METHOD PublishReceived : BOOL
  VAR_INPUT
    Data : MQTT.CALLBACK_DATA;  (* Collection of recived Data *)
  END_VAR
  VAR
    sSubTopic : STRING;
    NodeNumber : STRING;
    sNodeRegister : STRING;
    iWritePos : INT;  (* 1-based position of '/write/' within sSubTopic; 0 when it is absent. *)
  END_VAR
                  //first check if Mqtt is initialized, otherwise do nothing
IF NOT(bInitMqttDone) THEN
	//mark the interface call from the collector as done
	PublishReceived := TRUE;
//check if the packet is for this FB
ELSIF sMQTTSubscribeTopic = LEFT(Data.TopicOut^, LEN(sMQTTSubscribeTopic)) THEN
	//mark the interface call from the collector as done
	PublishReceived := TRUE;
	// process the data
	(* Parse by delimiter rather than by fixed width. The old code took the last
	   nine characters and then one character each for the node and the register,
	   so a command on '.../12/write/3' parsed as node 2 - a write silently aimed
	   at a different physical device. This block supports afbNodes 2..30. *)
	sSubTopic := RIGHT(Data.TopicOut^, LEN(Data.TopicOut^) - LEN(sMQTTSubscribeTopic));
	iWritePos := FIND(sSubTopic, '/write/');

	IF iWritePos >= 3 THEN
		// sSubTopic is '/<node>/write/<register>', so the node digits occupy
		// positions 2..iWritePos-1 and the register is everything past '/write/'.
		NodeNumber := MID(sSubTopic, iWritePos - 2, 2);
		sNodeRegister := RIGHT(sSubTopic, LEN(sSubTopic) - (iWritePos + 6));
	ELSE
		NodeNumber := '';
		sNodeRegister := '';
	END_IF

	(* A payload may be negative: -1 on a target register is how a Ducobox is told
	   to stop overriding and return to automatic, and the box's own target entity
	   is announced with a minimum of -1 for exactly that. The sign is taken off
	   before the digits are checked - so whether IS_NUM accepts a leading minus
	   does not matter - and put back through INT_TO_WORD, whose two's complement
	   is what the device reads back as -1. STRING_TO_WORD on '-1' does not. *)
	sPayload := Data.PayloadString^;
	bNegative := LEFT(sPayload, 1) = '-';
	IF bNegative THEN
		sDigits := RIGHT(sPayload, LEN(sPayload) - 1);
	ELSE
		sDigits := sPayload;
	END_IF

	IF iWritePos >= 3 AND
		OSCAT_BASIC.IS_NUM(NodeNumber) AND
		OSCAT_BASIC.IS_NUM(sNodeRegister) AND
		OSCAT_BASIC.IS_NUM(sDigits) AND
		(* 1 is the box itself, 2 and up are its components. The box is written
		   exactly like a component - its registers start at 10, which is what
		   index 1 gives - and InitMqttDiscovery announces three numbers and five
		   buttons for it. Requiring 2 here left every one of those controls inert,
		   and silently: falling through this guard looks identical to a topic
		   meant for some other device. *)
		STRING_TO_UINT(NodeNumber) >= 1 AND
		STRING_TO_UINT(NodeNumber) < THIS^.uiNodePointer THEN
			stWriteStep.Address := (STRING_TO_UINT(NodeNumber) * 10) + STRING_TO_UINT(sNodeRegister);
			IF bNegative THEN
				stWriteStep.Data[0] := INT_TO_WORD(-1 * STRING_TO_INT(sDigits));
			ELSE
				stWriteStep.Data[0] := STRING_TO_WORD(sDigits);
			END_IF
			sWriteQuerySuffix := sSubTopic;
			sWriteQueryPayload := Data.PayloadString^;
			bWriteQueryReady := TRUE;
	END_IF
END_IF
                
END_METHOD

METHOD AddNode : BOOL
  VAR_INPUT
    FriendlyName : STRING(GVL_MQTT.MQTT_SUFFIX_LEN);  (* Name of the room this component serves. *)
    DataPollingInterval : TIME;
  END_VAR
                  (* afbNodes is ARRAY[2..30]. Without this bound the 30th call wrote past the end of
   it, and the unassigned return value left the caller unable to notice. *)
IF uiNodePointer <= 30 THEN
	THIS^.afbNodes[uiNodePointer].InitNode(
		DeviceAddress := THIS^.stMasterStep.DeviceId,
		NodeNumber := uiNodePointer - 1,
		FriendlyName := FriendlyName,
		DataPollingInterval := DataPollingInterval
	);

	uiNodePointer := uiNodePointer + 1;
	AddNode := TRUE;
ELSE
	AddNode := FALSE;
END_IF

                
END_METHOD

METHOD BuildTransaction : INT
  VAR_INPUT
    pSteps : POINTER TO A_RS485_STEP_LIST;
  END_VAR
  VAR
    iN : INT;
    iK : INT;
    iI : INT;
  END_VAR
                  iN := 0;

IF bWriteQueryReady THEN
	bWriteQueryReady := FALSE;

	(* Write, then read the same register straight back, with the bus held
	   across both. What this block used to do was publish the payload it had
	   just sent, as though sending it were proof - so Home Assistant showed a
	   value the Ducobox might never have taken. AbortOnError on the write is
	   what stops the read-back running, and therefore stops anything being
	   published, when the write itself fails. *)
	pSteps^[iN]				:= stWriteStep;
	pSteps^[iN].AbortOnError	:= TRUE;
	aiStepMap[iN]				:= 2;
	iN						:= iN + 1;

	stReadBackStep.DeviceId		:= stWriteStep.DeviceId;
	(* Function 3: the register was written as a holding register, so that is
	   where it reads back from. If a Ducobox turns out to mirror these into the
	   input register space instead, this is the one line that changes. *)
	stReadBackStep.FunctionCode	:= 3;
	stReadBackStep.Address		:= stWriteStep.Address;
	stReadBackStep.Quantity		:= 1;

	pSteps^[iN]	:= stReadBackStep;
	aiStepMap[iN]	:= 3;
	iN			:= iN + 1;
END_IF

IF fbTimerData.Q THEN
	fbTimerData.IN	:= FALSE;
	pSteps^[iN]		:= stMasterStep;
	aiStepMap[iN]		:= 1;
	iN				:= iN + 1;
END_IF

(* One node per transaction, taken in turn from iNodeCursor. *)
FOR iK := 0 TO 28 DO
	iI := 2 + ((iNodeCursor - 2 + iK) MOD 29);
	IF iI < UINT_TO_INT(uiNodePointer) THEN
		IF afbNodes[iI].RequestBusTime() THEN
			pSteps^[iN]	:= afbNodes[iI].GetStep();
			aiStepMap[iN]	:= 10 + iI;
			iN			:= iN + 1;
			iNodeCursor	:= 2 + ((iI - 1) MOD 29);
			EXIT;
		END_IF
	END_IF
END_FOR

(* The zone read, at most one per transaction and only until each node has
   answered once. It rides behind the value read rather than competing with it,
   and it is a step of its own because read parameters 6..8 are undefined and the
   box rejects a span that crosses them. *)
FOR iK := 2 TO 30 DO
	IF iK < UINT_TO_INT(uiNodePointer) THEN
		IF afbNodes[iK].RequestLocation() THEN
			(* GetLocationStep answers with a zero-filled step if its retry clock
			   lapsed since RequestLocation was asked. Quantity 0 is not a Modbus
			   request: it fails locally, never reaches the bus, and so never shows
			   in the counters - while still counting as a failed step here. *)
			stLocStep := afbNodes[iK].GetLocationStep();
			IF stLocStep.Quantity > 0 THEN
				pSteps^[iN]	:= stLocStep;
				aiStepMap[iN]	:= 50 + iK;
				iN			:= iN + 1;
			END_IF
			EXIT;
		END_IF
	END_IF
END_FOR

(* One setting register per transaction, the box's own first. Deliberately
   last and one at a time: this is refresh traffic, it must never crowd out a
   command or a measurement, and reading a span would cross registers that are
   undefined on some component types. *)
IF bBoxSettingsDue THEN
	iBoxSettingsPending := -1;
	FOR iB := iBoxSettingsCursor TO 9 DO
		IF (wBoxSettingsMask AND SHL(WORD#1, INT_TO_BYTE(iB))) <> 0 THEN
			iBoxSettingsPending := iB;
			iBoxSettingsCursor := iB + 1;
			EXIT;
		END_IF
	END_FOR

	IF iBoxSettingsPending >= 0 THEN
		stBoxSettingsStep.Address := 10 + INT_TO_UINT(iBoxSettingsPending);
		pSteps^[iN]	:= stBoxSettingsStep;
		aiStepMap[iN]	:= 4;
		iN			:= iN + 1;
	ELSE
		bBoxSettingsDue := FALSE;
	END_IF
ELSE
	FOR iK := 2 TO 30 DO
		IF iK < UINT_TO_INT(uiNodePointer) THEN
			IF afbNodes[iK].RequestSettings() THEN
				stLocStep := afbNodes[iK].GetSettingsStep();
				IF stLocStep.Quantity > 0 THEN
					pSteps^[iN]	:= stLocStep;
					aiStepMap[iN]	:= 100 + iK;
					iN			:= iN + 1;
				END_IF
				EXIT;
			END_IF
		END_IF
	END_FOR
END_IF

(* Whether this transaction carried anything whose failure would really mean
   the box is unreachable: the master read, or a node's measurements. A lone
   zone read does not qualify. *)
bTxHadRequiredStep := FALSE;
FOR iK := 0 TO iN - 1 DO
	IF (aiStepMap[iK] = 1) OR ((aiStepMap[iK] >= 12) AND (aiStepMap[iK] <= 40)) THEN
		bTxHadRequiredStep := TRUE;
	END_IF
END_FOR

BuildTransaction := iN;

                
END_METHOD

METHOD HasWork : E_RS485_WORK_LEVEL
  VAR
    iK : INT;
  END_VAR
                  (* Pure predicate. afbNodes[].RequestBusTime is one too, so asking them here costs
   nothing and cannot disturb anything - which is the reason the node kept that
   method while the parent's own version was replaced. *)
IF NOT bInitRS485Done THEN
	HasWork := E_RS485_WORK_LEVEL.NONE;
	RETURN;
END_IF

IF bWriteQueryReady THEN
	(* Somebody is waiting on this: it arrived over MQTT, from Home Assistant or
	   a person. Ahead of routine polling, but still round-robin against other
	   devices' commands. *)
	HasWork := E_RS485_WORK_LEVEL.COMMAND;
	RETURN;
END_IF

IF fbTimerData.Q THEN
	HasWork := E_RS485_WORK_LEVEL.POLL;
	RETURN;
END_IF

IF bBoxSettingsDue THEN
	(* Refresh traffic, so it ranks with polling rather than with a command. *)
	HasWork := E_RS485_WORK_LEVEL.POLL;
	RETURN;
END_IF

HasWork := E_RS485_WORK_LEVEL.NONE;
FOR iK := 2 TO 30 DO
	IF iK < UINT_TO_INT(uiNodePointer) THEN
		(* RequestLocation counts as work: without it a node that has answered its
		   values but not its zone would never get another transaction built. *)
		IF afbNodes[iK].RequestBusTime() OR afbNodes[iK].RequestLocation()
			OR afbNodes[iK].RequestSettings() THEN
			HasWork := E_RS485_WORK_LEVEL.POLL;
			RETURN;
		END_IF
	END_IF
END_FOR

                
END_METHOD

METHOD OnStepResult
  VAR_INPUT
    StepIndex : INT;
    Failed : BOOL;
    pData : POINTER TO A_RS485_READ_BUFFER;
    Count : INT;
  END_VAR
  VAR
    iStepKind : INT;
  END_VAR
                  IF StepIndex < 0 OR StepIndex > DINT_TO_INT(UPPER_BOUND(aiStepMap, 1)) THEN
	RETURN;
END_IF

iStepKind := aiStepMap[StepIndex];

IF iStepKind = 1 THEN
	(* Master unit *)
	THIS^.Error := Failed;
	THIS^.fbTimerData.IN := TRUE;
	IF NOT Failed AND Count >= 6 THEN
		(* Publish only what moved. The box answers with the same six values poll
		   after poll - on the bench that was 126 identical messages in 100 seconds
		   against one or two from each node - and volume on this task is what made
		   the publish-queue race fire constantly before the queue got lanes.

		   Topics are not retained, so a value that never moves would never reach a
		   reconnecting Home Assistant; the refresh in the body forces a full
		   publish periodically regardless. *)
		bMasterChanged := NOT bMasterPublished OR bRefreshDue;
		FOR iMasterChk := 0 TO 5 DO
			IF pData^[iMasterChk] <> awLastMaster[iMasterChk] THEN
				bMasterChanged := TRUE;
			END_IF
			awLastMaster[iMasterChk] := pData^[iMasterChk];
		END_FOR

		IF bMasterChanged THEN
			bMasterPublished := TRUE;
			bRefreshDue := FALSE;
			PubMqttMessage(Suffix := '/1/TYPE', Data := F_DUCO_TYPE_TEXT(F_DUCO_NODE_TYPE(pData^[0])));
			PubMqttMessage(Suffix := '/1/STATUS', Data := F_DUCO_STATUS_TEXT(pData^[1]));
			PubMqttMessage(Suffix := '/1/POS', Data := WORD_TO_STRING(pData^[2]));
			(* Focus-specific: on this box read parameters 3, 4 and 5 are the current,
			   average and maximum power in watts. Another DucoBox answers the same
			   addresses with a different set, which is why this block is named. *)
			PubMqttMessage(Suffix := '/1/PWR', Data := WORD_TO_STRING(pData^[3]));
			PubMqttMessage(Suffix := '/1/PWR_AVG', Data := WORD_TO_STRING(pData^[4]));
			PubMqttMessage(Suffix := '/1/PWR_MAX', Data := WORD_TO_STRING(pData^[5]));
		END_IF
	END_IF

ELSIF iStepKind = 2 THEN
	(* The write. Deliberately publishes nothing: the value is only news once
	   the device has been read back and agrees. *)
	THIS^.Error := Failed;

ELSIF iStepKind = 3 THEN
	(* The read-back. This is the value the device actually holds, which is the
	   whole point of pairing the two. *)
	IF NOT Failed AND Count >= 1 THEN
		(* Suffix already begins with '/', so this leading one doubles it. Kept
		   as it was: the topic is what Home Assistant is already subscribed to,
		   and it cannot be re-checked without a Ducobox on the bench. *)
		(* One slash, not two. The suffix already begins with one, and the doubled
   topic was only harmless while nothing subscribed to it. The number and
   switch entities now take their state from here, so it has to be the topic
   their discovery config names. *)
PubMqttMessage(Suffix := sWriteQuerySuffix, Data := INT_TO_STRING(WORD_TO_INT(pData^[0])));
	END_IF

ELSIF iStepKind = 4 THEN
	(* The box's own setting, read back so its entity has a value before anybody
	   sets one. Signed for the same reason the write path is: -1 is a real
	   value here, meaning the box is not overriding. *)
	IF NOT Failed AND Count >= 1 AND iBoxSettingsPending >= 0 THEN
		PubMqttMessage(
			Suffix := CONCAT('/1/write/', INT_TO_STRING(iBoxSettingsPending)),
			Data := INT_TO_STRING(WORD_TO_INT(pData^[0])));
	END_IF
	iBoxSettingsPending := -1;

ELSIF iStepKind >= 12 AND iStepKind <= 40 THEN
	afbNodes[iStepKind - 10].OnStepResult(Failed := Failed, pData := pData, Count := Count);

ELSIF iStepKind >= 102 AND iStepKind <= 130 THEN
	(* 100 + node index: a setting register read back. A separate kind again,
	   because it lands in its own method and carries one register. *)
	afbNodes[iStepKind - 100].OnSettingsResult(Failed := Failed, pData := pData, Count := Count);

ELSIF iStepKind >= 52 AND iStepKind <= 80 THEN
	(* 50 + node index: the zone read. A separate kind from 10 + index because the
	   two steps carry different registers and land in different methods. *)
	afbNodes[iStepKind - 50].OnLocationResult(Failed := Failed, pData := pData, Count := Count);
END_IF

                
END_METHOD

METHOD OnTransactionDone
  VAR_INPUT
    StepsRun : INT;
    Failures : INT;
  END_VAR
                  (* Count, do not decide - and record what was actually seen.

   A single transaction is far too small a sample to condemn a device on: this
   bus interleaves the master read, one node's measurements, an optional zone
   read and any write that has arrived, and the mix differs every time. The
   verdict is taken on a heartbeat in the body instead. *)
uiTxCalls := uiTxCalls + 1;
iLastStepsRun := StepsRun;
iLastFailures := Failures;

IF StepsRun > 0 AND bTxHadRequiredStep THEN
	uiTxSeen := uiTxSeen + 1;
	IF Failures < StepsRun THEN
		uiTxOk := uiTxOk + 1;
	END_IF
END_IF

                
END_METHOD

(* Nothing to commission on this device. See I_RS485_DEVICE.GetCommissioning. *)
METHOD GetCommissioning : BOOL
  VAR_INPUT
    BusBaudrate : UDINT;
    pRequest : POINTER TO ST_RS485_COMMISSION_REQUEST;
  END_VAR
                  (* Nothing to commission. This device is configured on the device itself - switches,
   a display, or a factory setting that already matches this bus - so it answers at
   whatever the bus runs at and there is nothing for the commissioner to write.

   Which is the ordinary case: the cost of the whole mechanism, for a device like
   this one, is this method call once at bStartup. *)
GetCommissioning := FALSE;

                
END_METHOD

(* Announce the box and, as the bus reports what they are, every component on it. Call once at startup, after InitMqtt. *)
METHOD InitMqttDiscovery
  VAR_INPUT
    DeviceName : STRING(50);
    overruleId : STRING(255);
  END_VAR
  VAR
    sLabel : STRING(GVL_MQTT.MQTT_SUFFIX_LEN);
    sOut : STRING(GVL_MQTT.MQTT_TOPIC_LEN);
    sCmd : STRING(GVL_MQTT.MQTT_TOPIC_LEN);
  END_VAR
                  (* The box itself is node 1. Its own device; each component announces its own
   as the bus reports what it is, from the sweep in the body. *)
IF bInitMqttDone AND NOT bInitMqttDiscoveryDone THEN
	bInitMqttDiscoveryDone := TRUE;
	sDeviceId := SUPER^.ResolveEntityId(overruleId := overruleId);

	sLabel := DeviceName;
	sOut := CONCAT(THIS^.sMQTTPublishTopic, '/1');
	sCmd := CONCAT(THIS^.sMQTTSubscribeTopic, '/1');

	fbMqttDiscoveryDevice.initBaseDevice(
		Name := DeviceName,
		Identifiers := sDeviceId,
		Manufacturer := 'DUCO',
		Model := 'DucoBox Focus',
		availabilityTopic := GVL_MQTT.MqttAvailabilityTopic,
		availabilityTopic2 := CONCAT(THIS^.sMQTTPublishTopic, '/availability'),
		availabilityOnline := GVL_MQTT.MqttAvailabilityOnlinePayload,
		availabilityOffline := GVL_MQTT.MqttAvailabilityOfflinePayload,
		MqttDiscoveryPrefix := GVL_MQTT.MqttHADiscoveryPrefix,
		MqttDiagnosticTopic := CONCAT(THIS^.sMQTTPublishTopic, '/diagnostic'),
		pMqttPublishQueue := THIS^.pMqttPublishQueue);

(* This device publishes from the RS485 task, so its messages take that
   task's queue lane. A lane may only ever have one producing task. *)
fbMqttDiscoveryDevice.SetLane(Lane := GVL_MQTT.MQTT_LANE_RS485);

	fbMqttDiscoveryDevice.CreateSensorEntity(
		Name := CONCAT(sLabel, ' status'),
		Id := CONCAT(sDeviceId, '_STATUS'),
		StateTopic := CONCAT(sOut, '/STATUS'),
		ExpiryAfter := 0,
		DeviceClass := '',
		UnitOfMeasurement := '',
		StateClass := '',
		AvailabilityTopic := '');

	fbMqttDiscoveryDevice.CreateSensorEntity(
		Name := CONCAT(sLabel, ' ventilation position'),
		Id := CONCAT(sDeviceId, '_POS'),
		StateTopic := CONCAT(sOut, '/POS'),
		ExpiryAfter := 0,
		DeviceClass := '',
		UnitOfMeasurement := '%',
		StateClass := '',
		AvailabilityTopic := '');

	fbMqttDiscoveryDevice.CreateSensorEntity(
		Name := CONCAT(sLabel, ' power'),
		Id := CONCAT(sDeviceId, '_PWR'),
		StateTopic := CONCAT(sOut, '/PWR'),
		ExpiryAfter := 0,
		DeviceClass := 'power',
		UnitOfMeasurement := 'W',
		StateClass := 'measurement',
		AvailabilityTopic := '');

	fbMqttDiscoveryDevice.CreateSensorEntity(
		Name := CONCAT(sLabel, ' average power'),
		Id := CONCAT(sDeviceId, '_PWR_AVG'),
		StateTopic := CONCAT(sOut, '/PWR_AVG'),
		ExpiryAfter := 0,
		DeviceClass := 'power',
		UnitOfMeasurement := 'W',
		StateClass := 'measurement',
		AvailabilityTopic := '');

	fbMqttDiscoveryDevice.CreateSensorEntity(
		Name := CONCAT(sLabel, ' maximum power'),
		Id := CONCAT(sDeviceId, '_PWR_MAX'),
		StateTopic := CONCAT(sOut, '/PWR_MAX'),
		ExpiryAfter := 0,
		DeviceClass := 'power',
		UnitOfMeasurement := 'W',
		StateClass := 'measurement',
		AvailabilityTopic := '');

	fbMqttDiscoveryDevice.CreateNumberEntity(
		Name := CONCAT(sLabel, ' target'),
		Id := CONCAT(sDeviceId, '_W0'),
		CommandTopic := CONCAT(sCmd, '/write/0'),
		StateTopic := CONCAT(sOut, '/write/0'),
		MinValue := -1, MaxValue := 100, StepValue := 5,
		UnitOfMeasurement := '%', DeviceClass := '',
		EntityCategory := 'config', SliderMode := TRUE);

	fbMqttDiscoveryDevice.CreateNumberEntity(
		Name := CONCAT(sLabel, ' auto minimum'),
		Id := CONCAT(sDeviceId, '_W5'),
		CommandTopic := CONCAT(sCmd, '/write/5'),
		StateTopic := CONCAT(sOut, '/write/5'),
		MinValue := 0, MaxValue := 100, StepValue := 5,
		UnitOfMeasurement := '%', DeviceClass := '',
		EntityCategory := 'config', SliderMode := TRUE);

	fbMqttDiscoveryDevice.CreateNumberEntity(
		Name := CONCAT(sLabel, ' auto maximum'),
		Id := CONCAT(sDeviceId, '_W6'),
		CommandTopic := CONCAT(sCmd, '/write/6'),
		StateTopic := CONCAT(sOut, '/write/6'),
		MinValue := 0, MaxValue := 100, StepValue := 5,
		UnitOfMeasurement := '%', DeviceClass := '',
		EntityCategory := 'config', SliderMode := TRUE);

	(* Holding 9, the action. Buttons because the result is reported back under a
	   different encoding - status 4 is what action 2 produces - so a select would
	   have to be optimistic and would drift out of step.

	   Actions 2, 3 and 4 are TEMPORARY manual settings: the zone returns to
	   automatic on its own, after 15 minutes on an extraction system and 8 hours on
	   a supply one. The name says 'timed' rather than a number because the number
	   is not fixed - a room operating unit carries the duration in holding 7,
	   settable from 5 to 9995 minutes and announced here as its manual time
	   control. The box has no such register, and says nothing about the timer
	   either: the status it reports back is a plain 'Manual low', with no hint that
	   it lapses. Which is why the name has to carry that at all.

	   The 10, 20 and 30 minute high settings cannot be requested here. They exist
	   only as INPUT 1 status values, so a physical control can produce one and this
	   block can report it, but no action value asks for one. Holding 0, the target
	   percentage, is the other way to overrule - a level with no timer, already
	   exposed as the target number. *)
	fbMqttDiscoveryDevice.CreateButtonEntity(
		Name := CONCAT(sLabel, ' Low (timed)'),
		Id := CONCAT(sDeviceId, '_A2'),
		CommandTopic := CONCAT(sCmd, '/write/9'),
		PayloadPress := '2',
		EntityCategory := 'config', DeviceClass := '');

	fbMqttDiscoveryDevice.CreateButtonEntity(
		Name := CONCAT(sLabel, ' Medium (timed)'),
		Id := CONCAT(sDeviceId, '_A3'),
		CommandTopic := CONCAT(sCmd, '/write/9'),
		PayloadPress := '3',
		EntityCategory := 'config', DeviceClass := '');

	fbMqttDiscoveryDevice.CreateButtonEntity(
		Name := CONCAT(sLabel, ' High (timed)'),
		Id := CONCAT(sDeviceId, '_A4'),
		CommandTopic := CONCAT(sCmd, '/write/9'),
		PayloadPress := '4',
		EntityCategory := 'config', DeviceClass := '');

	fbMqttDiscoveryDevice.CreateButtonEntity(
		Name := CONCAT(sLabel, ' Auto'),
		Id := CONCAT(sDeviceId, '_A5'),
		CommandTopic := CONCAT(sCmd, '/write/9'),
		PayloadPress := '5',
		EntityCategory := 'config', DeviceClass := '');

	fbMqttDiscoveryDevice.CreateButtonEntity(
		Name := CONCAT(sLabel, ' Unoccupied'),
		Id := CONCAT(sDeviceId, '_A6'),
		CommandTopic := CONCAT(sCmd, '/write/9'),
		PayloadPress := '6',
		EntityCategory := 'config', DeviceClass := '');

END_IF
                
END_METHOD

(* Announce one component and everything its module type carries. *)
METHOD AnnounceNode
  VAR_INPUT
    iN : INT;
  END_VAR
  VAR
    eType : E_RS485_DUCO_NODE_TYPE;
    sNode : STRING(8);
    sLabel : STRING(GVL_MQTT.MQTT_SUFFIX_LEN);
    sId : STRING(255);
    sOut : STRING(GVL_MQTT.MQTT_TOPIC_LEN);
    sCmd : STRING(GVL_MQTT.MQTT_TOPIC_LEN);
    Device : POINTER TO FB_BASE_MQTT_DISCOVERY_DEVICE;
  END_VAR
                  Device := ADR(THIS^.fbMqttDiscoveryDevice);

(* One component, announced as a device of its own. The shared discovery object
   is re-pointed here and everything for this component is created before the
   next call re-points it again.

   The entity set comes from the module type read off the bus, not from anything
   declared at the call site - so a valve swapped for a sensor re-announces as a
   sensor without a code change. *)
eType := afbNodes[iN].GetNodeType();

IF eType = E_RS485_DUCO_NODE_TYPE.Unknown THEN
	RETURN;
END_IF

sNode  := UINT_TO_STRING(afbNodes[iN].GetNodeNumber());
sLabel := afbNodes[iN].GetFriendlyName();
sId    := CONCAT(CONCAT(sDeviceId, '_N'), sNode);
sOut   := CONCAT(CONCAT(THIS^.sMQTTPublishTopic, '/'), sNode);
sCmd    := CONCAT(CONCAT(THIS^.sMQTTSubscribeTopic, '/'), sNode);

Device^.initBaseDevice(
	Name := sLabel,
	Identifiers := sId,
	Manufacturer := 'DUCO',
	Model := F_DUCO_TYPE_TEXT(eType),
	availabilityTopic := GVL_MQTT.MqttAvailabilityTopic,
	availabilityTopic2 := CONCAT(THIS^.sMQTTPublishTopic, '/availability'),
	availabilityOnline := GVL_MQTT.MqttAvailabilityOnlinePayload,
	availabilityOffline := GVL_MQTT.MqttAvailabilityOfflinePayload,
	MqttDiscoveryPrefix := GVL_MQTT.MqttHADiscoveryPrefix,
	MqttDiagnosticTopic := CONCAT(THIS^.sMQTTPublishTopic, '/diagnostic'),
	pMqttPublishQueue := THIS^.pMqttPublishQueue);

(* This device publishes from the RS485 task, so its messages take that
   task's queue lane. A lane may only ever have one producing task. *)
Device^.SetLane(Lane := GVL_MQTT.MQTT_LANE_RS485);

(* Common to every component that has them. *)
Device^.CreateSensorEntity(
	Name := CONCAT(sLabel, ' status'),
	Id := CONCAT(sId, '_STATUS'),
	StateTopic := CONCAT(sOut, '/STATUS'),
	ExpiryAfter := 0,
	DeviceClass := '',
	UnitOfMeasurement := '',
	StateClass := '',
	AvailabilityTopic := '');

Device^.CreateSensorEntity(
	Name := CONCAT(sLabel, ' zone'),
	Id := CONCAT(sId, '_ZONE'),
	StateTopic := CONCAT(sOut, '/ZONE'),
	ExpiryAfter := 0,
	DeviceClass := '',
	UnitOfMeasurement := '',
	StateClass := '',
	AvailabilityTopic := '');

CASE eType OF

E_RS485_DUCO_NODE_TYPE.ValveSensorless,
E_RS485_DUCO_NODE_TYPE.ValveCO2,
E_RS485_DUCO_NODE_TYPE.ValveHumidity,
E_RS485_DUCO_NODE_TYPE.ValveHumidityCO2:
	Device^.CreateSensorEntity(
		Name := CONCAT(sLabel, ' position'),
		Id := CONCAT(sId, '_POS'),
		StateTopic := CONCAT(sOut, '/POS'),
		ExpiryAfter := 0,
		DeviceClass := '',
		UnitOfMeasurement := '%',
		StateClass := '',
		AvailabilityTopic := '');

	Device^.CreateSensorEntity(
		Name := CONCAT(sLabel, ' temperature'),
		Id := CONCAT(sId, '_TEMP'),
		StateTopic := CONCAT(sOut, '/TEMP'),
		ExpiryAfter := 0,
		DeviceClass := 'temperature',
		UnitOfMeasurement := '°C',
		StateClass := 'measurement',
		AvailabilityTopic := '');

	IF eType = E_RS485_DUCO_NODE_TYPE.ValveCO2 OR eType = E_RS485_DUCO_NODE_TYPE.ValveHumidityCO2 THEN
		Device^.CreateSensorEntity(
			Name := CONCAT(sLabel, ' CO2'),
			Id := CONCAT(sId, '_CO2'),
			StateTopic := CONCAT(sOut, '/CO2'),
			ExpiryAfter := 0,
			DeviceClass := 'carbon_dioxide',
			UnitOfMeasurement := 'ppm',
			StateClass := 'measurement',
			AvailabilityTopic := '');

		(* CO2 setpoint exists only where there is a CO2 sensor to compare it to. *)
		Device^.CreateNumberEntity(
			Name := CONCAT(sLabel, ' CO2 setpoint'),
			Id := CONCAT(sId, '_W1'),
			CommandTopic := CONCAT(sCmd, '/write/1'),
			StateTopic := CONCAT(sOut, '/write/1'),
			MinValue := 0, MaxValue := 2000, StepValue := 10,
			UnitOfMeasurement := 'ppm', DeviceClass := 'carbon_dioxide',
			EntityCategory := 'config', SliderMode := FALSE);

	END_IF
	IF eType = E_RS485_DUCO_NODE_TYPE.ValveHumidity OR eType = E_RS485_DUCO_NODE_TYPE.ValveHumidityCO2 THEN
		Device^.CreateSensorEntity(
			Name := CONCAT(sLabel, ' humidity'),
			Id := CONCAT(sId, '_RH'),
			StateTopic := CONCAT(sOut, '/RH'),
			ExpiryAfter := 0,
			DeviceClass := 'humidity',
			UnitOfMeasurement := '%',
			StateClass := 'measurement',
			AvailabilityTopic := '');

		Device^.CreateNumberEntity(
			Name := CONCAT(sLabel, ' humidity setpoint'),
			Id := CONCAT(sId, '_W2'),
			CommandTopic := CONCAT(sCmd, '/write/2'),
			StateTopic := CONCAT(sOut, '/write/2'),
			MinValue := 0, MaxValue := 100, StepValue := 5,
			UnitOfMeasurement := '%', DeviceClass := 'humidity',
			EntityCategory := 'config', SliderMode := TRUE);

		Device^.CreateSwitchEntity(
			Name := CONCAT(sLabel, ' humidity delta control'),
			Id := CONCAT(sId, '_W3'),
			CommandTopic := CONCAT(sCmd, '/write/3'),
			PayloadOn := '1', PayloadOff := '0',
			StateTopic := CONCAT(sOut, '/write/3'),
			StateOnPayload := '1', StateOffPayload := '0',
			DeviceClass := '');

	END_IF
	Device^.CreateNumberEntity(
		Name := CONCAT(sLabel, ' target'),
		Id := CONCAT(sId, '_W0'),
		CommandTopic := CONCAT(sCmd, '/write/0'),
		StateTopic := CONCAT(sOut, '/write/0'),
		MinValue := -1, MaxValue := 100, StepValue := 5,
		UnitOfMeasurement := '%', DeviceClass := '',
		EntityCategory := 'config', SliderMode := TRUE);

	Device^.CreateNumberEntity(
		Name := CONCAT(sLabel, ' flow'),
		Id := CONCAT(sId, '_W4'),
		CommandTopic := CONCAT(sCmd, '/write/4'),
		StateTopic := CONCAT(sOut, '/write/4'),
		MinValue := 20, MaxValue := 200, StepValue := 5,
		UnitOfMeasurement := 'm³/h', DeviceClass := '',
		EntityCategory := 'config', SliderMode := FALSE);

	Device^.CreateNumberEntity(
		Name := CONCAT(sLabel, ' auto minimum'),
		Id := CONCAT(sId, '_W5'),
		CommandTopic := CONCAT(sCmd, '/write/5'),
		StateTopic := CONCAT(sOut, '/write/5'),
		MinValue := 0, MaxValue := 100, StepValue := 5,
		UnitOfMeasurement := '%', DeviceClass := '',
		EntityCategory := 'config', SliderMode := TRUE);

	Device^.CreateNumberEntity(
		Name := CONCAT(sLabel, ' auto maximum'),
		Id := CONCAT(sId, '_W6'),
		CommandTopic := CONCAT(sCmd, '/write/6'),
		StateTopic := CONCAT(sOut, '/write/6'),
		MinValue := 0, MaxValue := 100, StepValue := 5,
		UnitOfMeasurement := '%', DeviceClass := '',
		EntityCategory := 'config', SliderMode := TRUE);

	(* The action parameter, holding 9. Buttons rather than a select: the result
	   is not readable back in the same encoding - the action that produces
	   'Manual low' is 2 and the status that reports it is 4 - so a select would
	   have to be optimistic and would drift. A button claims no state. *)
	Device^.CreateButtonEntity(
		Name := CONCAT(sLabel, ' Low (timed)'),
		Id := CONCAT(sId, '_A2'),
		CommandTopic := CONCAT(sCmd, '/write/9'),
		PayloadPress := '2',
		EntityCategory := 'config', DeviceClass := '');

	Device^.CreateButtonEntity(
		Name := CONCAT(sLabel, ' Medium (timed)'),
		Id := CONCAT(sId, '_A3'),
		CommandTopic := CONCAT(sCmd, '/write/9'),
		PayloadPress := '3',
		EntityCategory := 'config', DeviceClass := '');

	Device^.CreateButtonEntity(
		Name := CONCAT(sLabel, ' High (timed)'),
		Id := CONCAT(sId, '_A4'),
		CommandTopic := CONCAT(sCmd, '/write/9'),
		PayloadPress := '4',
		EntityCategory := 'config', DeviceClass := '');

	Device^.CreateButtonEntity(
		Name := CONCAT(sLabel, ' Auto'),
		Id := CONCAT(sId, '_A5'),
		CommandTopic := CONCAT(sCmd, '/write/9'),
		PayloadPress := '5',
		EntityCategory := 'config', DeviceClass := '');

	Device^.CreateButtonEntity(
		Name := CONCAT(sLabel, ' Unoccupied'),
		Id := CONCAT(sId, '_A6'),
		CommandTopic := CONCAT(sCmd, '/write/9'),
		PayloadPress := '6',
		EntityCategory := 'config', DeviceClass := '');

E_RS485_DUCO_NODE_TYPE.UserControl:
	Device^.CreateSensorEntity(
		Name := CONCAT(sLabel, ' position'),
		Id := CONCAT(sId, '_POS'),
		StateTopic := CONCAT(sOut, '/POS'),
		ExpiryAfter := 0,
		DeviceClass := '',
		UnitOfMeasurement := '%',
		StateClass := '',
		AvailabilityTopic := '');

	Device^.CreateSensorEntity(
		Name := CONCAT(sLabel, ' temperature'),
		Id := CONCAT(sId, '_TEMP'),
		StateTopic := CONCAT(sOut, '/TEMP'),
		ExpiryAfter := 0,
		DeviceClass := 'temperature',
		UnitOfMeasurement := '°C',
		StateClass := 'measurement',
		AvailabilityTopic := '');

	Device^.CreateNumberEntity(
		Name := CONCAT(sLabel, ' target'),
		Id := CONCAT(sId, '_W0'),
		CommandTopic := CONCAT(sCmd, '/write/0'),
		StateTopic := CONCAT(sOut, '/write/0'),
		MinValue := -1, MaxValue := 100, StepValue := 5,
		UnitOfMeasurement := '%', DeviceClass := '',
		EntityCategory := 'config', SliderMode := TRUE);

	(* Holding 5 and 6 are the button values on a wall control, NOT auto min and
	   max as they are on a valve. Writing them as auto limits would retune
	   somebody's switch. *)
	Device^.CreateNumberEntity(
		Name := CONCAT(sLabel, ' button 1'),
		Id := CONCAT(sId, '_W4'),
		CommandTopic := CONCAT(sCmd, '/write/4'),
		StateTopic := CONCAT(sOut, '/write/4'),
		MinValue := 0, MaxValue := 100, StepValue := 5,
		UnitOfMeasurement := '%', DeviceClass := '',
		EntityCategory := 'config', SliderMode := TRUE);

	Device^.CreateNumberEntity(
		Name := CONCAT(sLabel, ' button 2'),
		Id := CONCAT(sId, '_W5'),
		CommandTopic := CONCAT(sCmd, '/write/5'),
		StateTopic := CONCAT(sOut, '/write/5'),
		MinValue := 0, MaxValue := 100, StepValue := 5,
		UnitOfMeasurement := '%', DeviceClass := '',
		EntityCategory := 'config', SliderMode := TRUE);

	Device^.CreateNumberEntity(
		Name := CONCAT(sLabel, ' button 3'),
		Id := CONCAT(sId, '_W6'),
		CommandTopic := CONCAT(sCmd, '/write/6'),
		StateTopic := CONCAT(sOut, '/write/6'),
		MinValue := 0, MaxValue := 100, StepValue := 5,
		UnitOfMeasurement := '%', DeviceClass := '',
		EntityCategory := 'config', SliderMode := TRUE);

	Device^.CreateNumberEntity(
		Name := CONCAT(sLabel, ' manual time'),
		Id := CONCAT(sId, '_W7'),
		CommandTopic := CONCAT(sCmd, '/write/7'),
		StateTopic := CONCAT(sOut, '/write/7'),
		MinValue := 5, MaxValue := 9995, StepValue := 5,
		UnitOfMeasurement := 'min', DeviceClass := '',
		EntityCategory := 'config', SliderMode := FALSE);

	(* The action parameter, holding 9. Buttons rather than a select: the result
	   is not readable back in the same encoding - the action that produces
	   'Manual low' is 2 and the status that reports it is 4 - so a select would
	   have to be optimistic and would drift. A button claims no state. *)
	Device^.CreateButtonEntity(
		Name := CONCAT(sLabel, ' Low (timed)'),
		Id := CONCAT(sId, '_A2'),
		CommandTopic := CONCAT(sCmd, '/write/9'),
		PayloadPress := '2',
		EntityCategory := 'config', DeviceClass := '');

	Device^.CreateButtonEntity(
		Name := CONCAT(sLabel, ' Medium (timed)'),
		Id := CONCAT(sId, '_A3'),
		CommandTopic := CONCAT(sCmd, '/write/9'),
		PayloadPress := '3',
		EntityCategory := 'config', DeviceClass := '');

	Device^.CreateButtonEntity(
		Name := CONCAT(sLabel, ' High (timed)'),
		Id := CONCAT(sId, '_A4'),
		CommandTopic := CONCAT(sCmd, '/write/9'),
		PayloadPress := '4',
		EntityCategory := 'config', DeviceClass := '');

	Device^.CreateButtonEntity(
		Name := CONCAT(sLabel, ' Auto'),
		Id := CONCAT(sId, '_A5'),
		CommandTopic := CONCAT(sCmd, '/write/9'),
		PayloadPress := '5',
		EntityCategory := 'config', DeviceClass := '');

	Device^.CreateButtonEntity(
		Name := CONCAT(sLabel, ' Unoccupied'),
		Id := CONCAT(sId, '_A6'),
		CommandTopic := CONCAT(sCmd, '/write/9'),
		PayloadPress := '6',
		EntityCategory := 'config', DeviceClass := '');

E_RS485_DUCO_NODE_TYPE.SensorCO2:
	Device^.CreateSensorEntity(
		Name := CONCAT(sLabel, ' temperature'),
		Id := CONCAT(sId, '_TEMP'),
		StateTopic := CONCAT(sOut, '/TEMP'),
		ExpiryAfter := 0,
		DeviceClass := 'temperature',
		UnitOfMeasurement := '°C',
		StateClass := 'measurement',
		AvailabilityTopic := '');

	Device^.CreateSensorEntity(
		Name := CONCAT(sLabel, ' CO2'),
		Id := CONCAT(sId, '_CO2'),
		StateTopic := CONCAT(sOut, '/CO2'),
		ExpiryAfter := 0,
		DeviceClass := 'carbon_dioxide',
		UnitOfMeasurement := 'ppm',
		StateClass := 'measurement',
		AvailabilityTopic := '');

	Device^.CreateNumberEntity(
		Name := CONCAT(sLabel, ' target'),
		Id := CONCAT(sId, '_W0'),
		CommandTopic := CONCAT(sCmd, '/write/0'),
		StateTopic := CONCAT(sOut, '/write/0'),
		MinValue := -1, MaxValue := 100, StepValue := 5,
		UnitOfMeasurement := '%', DeviceClass := '',
		EntityCategory := 'config', SliderMode := TRUE);

	Device^.CreateNumberEntity(
		Name := CONCAT(sLabel, ' CO2 setpoint'),
		Id := CONCAT(sId, '_W1'),
		CommandTopic := CONCAT(sCmd, '/write/1'),
		StateTopic := CONCAT(sOut, '/write/1'),
		MinValue := 0, MaxValue := 2000, StepValue := 10,
		UnitOfMeasurement := 'ppm', DeviceClass := 'carbon_dioxide',
		EntityCategory := 'config', SliderMode := FALSE);

	(* The action parameter, holding 9. Buttons rather than a select: the result
	   is not readable back in the same encoding - the action that produces
	   'Manual low' is 2 and the status that reports it is 4 - so a select would
	   have to be optimistic and would drift. A button claims no state. *)
	Device^.CreateButtonEntity(
		Name := CONCAT(sLabel, ' Low (timed)'),
		Id := CONCAT(sId, '_A2'),
		CommandTopic := CONCAT(sCmd, '/write/9'),
		PayloadPress := '2',
		EntityCategory := 'config', DeviceClass := '');

	Device^.CreateButtonEntity(
		Name := CONCAT(sLabel, ' Medium (timed)'),
		Id := CONCAT(sId, '_A3'),
		CommandTopic := CONCAT(sCmd, '/write/9'),
		PayloadPress := '3',
		EntityCategory := 'config', DeviceClass := '');

	Device^.CreateButtonEntity(
		Name := CONCAT(sLabel, ' High (timed)'),
		Id := CONCAT(sId, '_A4'),
		CommandTopic := CONCAT(sCmd, '/write/9'),
		PayloadPress := '4',
		EntityCategory := 'config', DeviceClass := '');

	Device^.CreateButtonEntity(
		Name := CONCAT(sLabel, ' Auto'),
		Id := CONCAT(sId, '_A5'),
		CommandTopic := CONCAT(sCmd, '/write/9'),
		PayloadPress := '5',
		EntityCategory := 'config', DeviceClass := '');

	Device^.CreateButtonEntity(
		Name := CONCAT(sLabel, ' Unoccupied'),
		Id := CONCAT(sId, '_A6'),
		CommandTopic := CONCAT(sCmd, '/write/9'),
		PayloadPress := '6',
		EntityCategory := 'config', DeviceClass := '');

E_RS485_DUCO_NODE_TYPE.SensorHumidity:
	Device^.CreateSensorEntity(
		Name := CONCAT(sLabel, ' temperature'),
		Id := CONCAT(sId, '_TEMP'),
		StateTopic := CONCAT(sOut, '/TEMP'),
		ExpiryAfter := 0,
		DeviceClass := 'temperature',
		UnitOfMeasurement := '°C',
		StateClass := 'measurement',
		AvailabilityTopic := '');

	Device^.CreateSensorEntity(
		Name := CONCAT(sLabel, ' humidity'),
		Id := CONCAT(sId, '_RH'),
		StateTopic := CONCAT(sOut, '/RH'),
		ExpiryAfter := 0,
		DeviceClass := 'humidity',
		UnitOfMeasurement := '%',
		StateClass := 'measurement',
		AvailabilityTopic := '');

	Device^.CreateNumberEntity(
		Name := CONCAT(sLabel, ' target'),
		Id := CONCAT(sId, '_W0'),
		CommandTopic := CONCAT(sCmd, '/write/0'),
		StateTopic := CONCAT(sOut, '/write/0'),
		MinValue := -1, MaxValue := 100, StepValue := 5,
		UnitOfMeasurement := '%', DeviceClass := '',
		EntityCategory := 'config', SliderMode := TRUE);

	Device^.CreateNumberEntity(
		Name := CONCAT(sLabel, ' humidity setpoint'),
		Id := CONCAT(sId, '_W2'),
		CommandTopic := CONCAT(sCmd, '/write/2'),
		StateTopic := CONCAT(sOut, '/write/2'),
		MinValue := 0, MaxValue := 100, StepValue := 5,
		UnitOfMeasurement := '%', DeviceClass := 'humidity',
		EntityCategory := 'config', SliderMode := TRUE);

	Device^.CreateSwitchEntity(
		Name := CONCAT(sLabel, ' humidity delta control'),
		Id := CONCAT(sId, '_W3'),
		CommandTopic := CONCAT(sCmd, '/write/3'),
		PayloadOn := '1', PayloadOff := '0',
		StateTopic := CONCAT(sOut, '/write/3'),
		StateOnPayload := '1', StateOffPayload := '0',
		DeviceClass := '');

	(* The action parameter, holding 9. Buttons rather than a select: the result
	   is not readable back in the same encoding - the action that produces
	   'Manual low' is 2 and the status that reports it is 4 - so a select would
	   have to be optimistic and would drift. A button claims no state. *)
	Device^.CreateButtonEntity(
		Name := CONCAT(sLabel, ' Low (timed)'),
		Id := CONCAT(sId, '_A2'),
		CommandTopic := CONCAT(sCmd, '/write/9'),
		PayloadPress := '2',
		EntityCategory := 'config', DeviceClass := '');

	Device^.CreateButtonEntity(
		Name := CONCAT(sLabel, ' Medium (timed)'),
		Id := CONCAT(sId, '_A3'),
		CommandTopic := CONCAT(sCmd, '/write/9'),
		PayloadPress := '3',
		EntityCategory := 'config', DeviceClass := '');

	Device^.CreateButtonEntity(
		Name := CONCAT(sLabel, ' High (timed)'),
		Id := CONCAT(sId, '_A4'),
		CommandTopic := CONCAT(sCmd, '/write/9'),
		PayloadPress := '4',
		EntityCategory := 'config', DeviceClass := '');

	Device^.CreateButtonEntity(
		Name := CONCAT(sLabel, ' Auto'),
		Id := CONCAT(sId, '_A5'),
		CommandTopic := CONCAT(sCmd, '/write/9'),
		PayloadPress := '5',
		EntityCategory := 'config', DeviceClass := '');

	Device^.CreateButtonEntity(
		Name := CONCAT(sLabel, ' Unoccupied'),
		Id := CONCAT(sId, '_A6'),
		CommandTopic := CONCAT(sCmd, '/write/9'),
		PayloadPress := '6',
		EntityCategory := 'config', DeviceClass := '');

E_RS485_DUCO_NODE_TYPE.WindowVentilator:
	Device^.CreateSensorEntity(
		Name := CONCAT(sLabel, ' opening'),
		Id := CONCAT(sId, '_OPEN'),
		StateTopic := CONCAT(sOut, '/OPEN'),
		ExpiryAfter := 0,
		DeviceClass := '',
		UnitOfMeasurement := '%',
		StateClass := '',
		AvailabilityTopic := '');

	Device^.CreateSensorEntity(
		Name := CONCAT(sLabel, ' outdoor temperature'),
		Id := CONCAT(sId, '_TEMP_OUT'),
		StateTopic := CONCAT(sOut, '/TEMP_OUT'),
		ExpiryAfter := 0,
		DeviceClass := 'temperature',
		UnitOfMeasurement := '°C',
		StateClass := 'measurement',
		AvailabilityTopic := '');

	Device^.CreateNumberEntity(
		Name := CONCAT(sLabel, ' target'),
		Id := CONCAT(sId, '_W0'),
		CommandTopic := CONCAT(sCmd, '/write/0'),
		StateTopic := CONCAT(sOut, '/write/0'),
		MinValue := -1, MaxValue := 100, StepValue := 5,
		UnitOfMeasurement := '%', DeviceClass := '',
		EntityCategory := 'config', SliderMode := TRUE);

	Device^.CreateNumberEntity(
		Name := CONCAT(sLabel, ' inlet share'),
		Id := CONCAT(sId, '_W4'),
		CommandTopic := CONCAT(sCmd, '/write/4'),
		StateTopic := CONCAT(sOut, '/write/4'),
		MinValue := 0, MaxValue := 100, StepValue := 5,
		UnitOfMeasurement := '%', DeviceClass := '',
		EntityCategory := 'config', SliderMode := TRUE);

	Device^.CreateNumberEntity(
		Name := CONCAT(sLabel, ' auto minimum'),
		Id := CONCAT(sId, '_W5'),
		CommandTopic := CONCAT(sCmd, '/write/5'),
		StateTopic := CONCAT(sOut, '/write/5'),
		MinValue := 0, MaxValue := 100, StepValue := 5,
		UnitOfMeasurement := '%', DeviceClass := '',
		EntityCategory := 'config', SliderMode := TRUE);

	Device^.CreateNumberEntity(
		Name := CONCAT(sLabel, ' auto maximum'),
		Id := CONCAT(sId, '_W6'),
		CommandTopic := CONCAT(sCmd, '/write/6'),
		StateTopic := CONCAT(sOut, '/write/6'),
		MinValue := 0, MaxValue := 100, StepValue := 5,
		UnitOfMeasurement := '%', DeviceClass := '',
		EntityCategory := 'config', SliderMode := TRUE);

	(* The action parameter, holding 9. Buttons rather than a select: the result
	   is not readable back in the same encoding - the action that produces
	   'Manual low' is 2 and the status that reports it is 4 - so a select would
	   have to be optimistic and would drift. A button claims no state. *)
	Device^.CreateButtonEntity(
		Name := CONCAT(sLabel, ' Low (timed)'),
		Id := CONCAT(sId, '_A2'),
		CommandTopic := CONCAT(sCmd, '/write/9'),
		PayloadPress := '2',
		EntityCategory := 'config', DeviceClass := '');

	Device^.CreateButtonEntity(
		Name := CONCAT(sLabel, ' Medium (timed)'),
		Id := CONCAT(sId, '_A3'),
		CommandTopic := CONCAT(sCmd, '/write/9'),
		PayloadPress := '3',
		EntityCategory := 'config', DeviceClass := '');

	Device^.CreateButtonEntity(
		Name := CONCAT(sLabel, ' High (timed)'),
		Id := CONCAT(sId, '_A4'),
		CommandTopic := CONCAT(sCmd, '/write/9'),
		PayloadPress := '4',
		EntityCategory := 'config', DeviceClass := '');

	Device^.CreateButtonEntity(
		Name := CONCAT(sLabel, ' Auto'),
		Id := CONCAT(sId, '_A5'),
		CommandTopic := CONCAT(sCmd, '/write/9'),
		PayloadPress := '5',
		EntityCategory := 'config', DeviceClass := '');

	Device^.CreateButtonEntity(
		Name := CONCAT(sLabel, ' Unoccupied'),
		Id := CONCAT(sId, '_A6'),
		CommandTopic := CONCAT(sCmd, '/write/9'),
		PayloadPress := '6',
		EntityCategory := 'config', DeviceClass := '');

E_RS485_DUCO_NODE_TYPE.SwitchSensor:
	Device^.CreateSensorEntity(
		Name := CONCAT(sLabel, ' position'),
		Id := CONCAT(sId, '_POS'),
		StateTopic := CONCAT(sOut, '/POS'),
		ExpiryAfter := 0,
		DeviceClass := '',
		UnitOfMeasurement := '%',
		StateClass := '',
		AvailabilityTopic := '');

	Device^.CreateNumberEntity(
		Name := CONCAT(sLabel, ' target'),
		Id := CONCAT(sId, '_W0'),
		CommandTopic := CONCAT(sCmd, '/write/0'),
		StateTopic := CONCAT(sOut, '/write/0'),
		MinValue := -1, MaxValue := 100, StepValue := 5,
		UnitOfMeasurement := '%', DeviceClass := '',
		EntityCategory := 'config', SliderMode := TRUE);

	(* Switch mode: 0 overrule, 1 heat pump, 2 presence. A number rather than a
	   select, because a select needs an options array and the JSON composer
	   cannot build one from this struct shape. *)
	Device^.CreateNumberEntity(
		Name := CONCAT(sLabel, ' switch mode'),
		Id := CONCAT(sId, '_W1'),
		CommandTopic := CONCAT(sCmd, '/write/1'),
		StateTopic := CONCAT(sOut, '/write/1'),
		MinValue := 0, MaxValue := 2, StepValue := 1,
		UnitOfMeasurement := '', DeviceClass := '',
		EntityCategory := 'config', SliderMode := FALSE);

	Device^.CreateNumberEntity(
		Name := CONCAT(sLabel, ' switch value'),
		Id := CONCAT(sId, '_W2'),
		CommandTopic := CONCAT(sCmd, '/write/2'),
		StateTopic := CONCAT(sOut, '/write/2'),
		MinValue := 0, MaxValue := 255, StepValue := 5,
		UnitOfMeasurement := '', DeviceClass := '',
		EntityCategory := 'config', SliderMode := FALSE);

	(* The action parameter, holding 9. Buttons rather than a select: the result
	   is not readable back in the same encoding - the action that produces
	   'Manual low' is 2 and the status that reports it is 4 - so a select would
	   have to be optimistic and would drift. A button claims no state. *)
	Device^.CreateButtonEntity(
		Name := CONCAT(sLabel, ' Low (timed)'),
		Id := CONCAT(sId, '_A2'),
		CommandTopic := CONCAT(sCmd, '/write/9'),
		PayloadPress := '2',
		EntityCategory := 'config', DeviceClass := '');

	Device^.CreateButtonEntity(
		Name := CONCAT(sLabel, ' Medium (timed)'),
		Id := CONCAT(sId, '_A3'),
		CommandTopic := CONCAT(sCmd, '/write/9'),
		PayloadPress := '3',
		EntityCategory := 'config', DeviceClass := '');

	Device^.CreateButtonEntity(
		Name := CONCAT(sLabel, ' High (timed)'),
		Id := CONCAT(sId, '_A4'),
		CommandTopic := CONCAT(sCmd, '/write/9'),
		PayloadPress := '4',
		EntityCategory := 'config', DeviceClass := '');

	Device^.CreateButtonEntity(
		Name := CONCAT(sLabel, ' Auto'),
		Id := CONCAT(sId, '_A5'),
		CommandTopic := CONCAT(sCmd, '/write/9'),
		PayloadPress := '5',
		EntityCategory := 'config', DeviceClass := '');

	Device^.CreateButtonEntity(
		Name := CONCAT(sLabel, ' Unoccupied'),
		Id := CONCAT(sId, '_A6'),
		CommandTopic := CONCAT(sCmd, '/write/9'),
		PayloadPress := '6',
		EntityCategory := 'config', DeviceClass := '');

E_RS485_DUCO_NODE_TYPE.ActuatorBoard:
	Device^.CreateSensorEntity(
		Name := CONCAT(sLabel, ' position'),
		Id := CONCAT(sId, '_POS'),
		StateTopic := CONCAT(sOut, '/POS'),
		ExpiryAfter := 0,
		DeviceClass := '',
		UnitOfMeasurement := '%',
		StateClass := '',
		AvailabilityTopic := '');

	Device^.CreateSensorEntity(
		Name := CONCAT(sLabel, ' outdoor temperature'),
		Id := CONCAT(sId, '_TEMP_OUT'),
		StateTopic := CONCAT(sOut, '/TEMP_OUT'),
		ExpiryAfter := 0,
		DeviceClass := 'temperature',
		UnitOfMeasurement := '°C',
		StateClass := 'measurement',
		AvailabilityTopic := '');

	Device^.CreateSensorEntity(
		Name := CONCAT(sLabel, ' PWM input'),
		Id := CONCAT(sId, '_PWM'),
		StateTopic := CONCAT(sOut, '/PWM'),
		ExpiryAfter := 0,
		DeviceClass := '',
		UnitOfMeasurement := '%',
		StateClass := '',
		AvailabilityTopic := '');

	Device^.CreateNumberEntity(
		Name := CONCAT(sLabel, ' target'),
		Id := CONCAT(sId, '_W0'),
		CommandTopic := CONCAT(sCmd, '/write/0'),
		StateTopic := CONCAT(sOut, '/write/0'),
		MinValue := -1, MaxValue := 100, StepValue := 5,
		UnitOfMeasurement := '%', DeviceClass := '',
		EntityCategory := 'config', SliderMode := TRUE);

	Device^.CreateNumberEntity(
		Name := CONCAT(sLabel, ' hybrid value'),
		Id := CONCAT(sId, '_W1'),
		CommandTopic := CONCAT(sCmd, '/write/1'),
		StateTopic := CONCAT(sOut, '/write/1'),
		MinValue := 0, MaxValue := 100, StepValue := 5,
		UnitOfMeasurement := '%', DeviceClass := '',
		EntityCategory := 'config', SliderMode := TRUE);

	Device^.CreateNumberEntity(
		Name := CONCAT(sLabel, ' inlet share'),
		Id := CONCAT(sId, '_W4'),
		CommandTopic := CONCAT(sCmd, '/write/4'),
		StateTopic := CONCAT(sOut, '/write/4'),
		MinValue := 0, MaxValue := 100, StepValue := 5,
		UnitOfMeasurement := '%', DeviceClass := '',
		EntityCategory := 'config', SliderMode := TRUE);

	Device^.CreateNumberEntity(
		Name := CONCAT(sLabel, ' auto minimum'),
		Id := CONCAT(sId, '_W5'),
		CommandTopic := CONCAT(sCmd, '/write/5'),
		StateTopic := CONCAT(sOut, '/write/5'),
		MinValue := 0, MaxValue := 100, StepValue := 5,
		UnitOfMeasurement := '%', DeviceClass := '',
		EntityCategory := 'config', SliderMode := TRUE);

	Device^.CreateNumberEntity(
		Name := CONCAT(sLabel, ' auto maximum'),
		Id := CONCAT(sId, '_W6'),
		CommandTopic := CONCAT(sCmd, '/write/6'),
		StateTopic := CONCAT(sOut, '/write/6'),
		MinValue := 0, MaxValue := 100, StepValue := 5,
		UnitOfMeasurement := '%', DeviceClass := '',
		EntityCategory := 'config', SliderMode := TRUE);

	(* The action parameter, holding 9. Buttons rather than a select: the result
	   is not readable back in the same encoding - the action that produces
	   'Manual low' is 2 and the status that reports it is 4 - so a select would
	   have to be optimistic and would drift. A button claims no state. *)
	Device^.CreateButtonEntity(
		Name := CONCAT(sLabel, ' Low (timed)'),
		Id := CONCAT(sId, '_A2'),
		CommandTopic := CONCAT(sCmd, '/write/9'),
		PayloadPress := '2',
		EntityCategory := 'config', DeviceClass := '');

	Device^.CreateButtonEntity(
		Name := CONCAT(sLabel, ' Medium (timed)'),
		Id := CONCAT(sId, '_A3'),
		CommandTopic := CONCAT(sCmd, '/write/9'),
		PayloadPress := '3',
		EntityCategory := 'config', DeviceClass := '');

	Device^.CreateButtonEntity(
		Name := CONCAT(sLabel, ' High (timed)'),
		Id := CONCAT(sId, '_A4'),
		CommandTopic := CONCAT(sCmd, '/write/9'),
		PayloadPress := '4',
		EntityCategory := 'config', DeviceClass := '');

	Device^.CreateButtonEntity(
		Name := CONCAT(sLabel, ' Auto'),
		Id := CONCAT(sId, '_A5'),
		CommandTopic := CONCAT(sCmd, '/write/9'),
		PayloadPress := '5',
		EntityCategory := 'config', DeviceClass := '');

	Device^.CreateButtonEntity(
		Name := CONCAT(sLabel, ' Unoccupied'),
		Id := CONCAT(sId, '_A6'),
		CommandTopic := CONCAT(sCmd, '/write/9'),
		PayloadPress := '6',
		EntityCategory := 'config', DeviceClass := '');

END_CASE

afbNodes[iN].SetAnnounced();
                
END_METHOD

(* Publish the device availability, retained. *)
METHOD PubAvailability
  VAR_INPUT
    Online : BOOL;
  END_VAR
                  (* Retained, unlike everything else this block publishes.

   Availability is device state, not an event: without the retain flag Home
   Assistant has nothing at all after any broker reconnect and greys out every
   entity of this device until the next heartbeat. The PLC's own availability
   topic is the second entry in the discovery config's avty list and carries the
   last will, so a controller that dies still marks these offline. *)
uiAvailPubs := uiAvailPubs + 1;

IF bInitMqttDone THEN
	IF Online THEN
		pMqttPublishQueue^.AddMessageOn(Lane := GVL_MQTT.MQTT_LANE_RS485,
			Payload := 'online',
			Topic := CONCAT(THIS^.sMQTTPublishTopic, '/availability'),
			Qos := MQTT.QoS.ExactlyOnce,
			MqttRetain := TRUE);
	ELSE
		pMqttPublishQueue^.AddMessageOn(Lane := GVL_MQTT.MQTT_LANE_RS485,
			Payload := 'offline',
			Topic := CONCAT(THIS^.sMQTTPublishTopic, '/availability'),
			Qos := MQTT.QoS.ExactlyOnce,
			MqttRetain := TRUE);
	END_IF
END_IF

                
END_METHOD
END_FUNCTION_BLOCK

FUNCTION_BLOCK FB_RS485_DUCO_DUCOBOX_FOCUS_NODE_MQTT
  VAR
    NodeNumber : UINT;
    bInitMqttDone : BOOL;
    psMqttPublishTopicPrefix : POINTER TO STRING;
    MqttPublishTopicSuffix : STRING(GVL_MQTT.MQTT_SUFFIX_LEN);
    pMqttPublishQueue : POINTER TO FB_MQTT_PUBLISH_QUEUE;
    bNodeInitialized : BOOL := FALSE;
    fbTimerData : TON;
    stStep : ST_RS485_STEP;  (* This node's read block. Filled by InitNode in code; a node is not registered on the bus in its own right, its parent puts this stStep into the transaction it builds. *)
    eType : E_RS485_DUCO_NODE_TYPE;  (* What this node is, decoded from read parameter 0 on the first successful read. Unknown until then, and Unknown again if the bus starts answering with a type this project does not name - which is a state worth having, because a component whose register layout is unknown must not get labelled entities. *)
    FriendlyName : STRING(GVL_MQTT.MQTT_SUFFIX_LEN);  (* The room, supplied by the call site. The MQTT topic still uses the node number: a topic that moved when somebody renamed a room would orphan its own retained state. *)
    stLocationStep : ST_RS485_STEP;  (* Read parameter 9, the zone grouping. Its own step, because parameters 6, 7 and 8 are undefined on every component type in L8000009 and a span of ten crosses them - the box answers that with an exception, not with zeroes. Read once when the node is first identified and then left alone. It changes only when the network is re-paired, so polling it would double this node's frames for a value that never moves. *)
    fbLocationRetry : TON;  (* Retry clock for the zone read. It replaces a wanted/known pair that could not recover: the request was cleared when the step was built and only a result put it back, so one result that never arrived lost the zone for the life of the application. A clock cannot get stuck that way - it simply asks again. *)
    bLocationKnown : BOOL := FALSE;
    bAnnounced : BOOL := FALSE;  (* Cleared when the module type changes, so a re-paired network re-announces rather than leaving Home Assistant describing the component that used to be at this node number. *)
    uiLocationTries : UINT := 0;  (* A box that will not answer read parameter 9 is not going to start. Three attempts, then the zone is simply not published - better than asking forever and putting a failing step on the bus every thirty seconds. *)
    awLastRaw : ARRAY[0..5] OF WORD;  (* Last raw frame, so unchanged values are not republished. A Duco reading moves rarely and the RS485 task was putting five topics per node into the publish queue every poll regardless - which is what made a latent race in that queue fire constantly. *)
    bPublishedOnce : BOOL := FALSE;
    bRefreshDue : BOOL := TRUE;
    iChk : INT;
    bChanged : BOOL;
    fbRepublish : TON;
    wSettingsMask : WORD := 0;  (* Which of this component's registers carry a setting Home Assistant shows, one bit per register, and where the refresh sweep has got to. See SettingsMaskFor. *)
    iSettingsCursor : INT := 0;
    iSettingsPending : INT := -1;
    bSettingsDue : BOOL := FALSE;
    stSettingsStep : ST_RS485_STEP;
    iS : INT;
  END_VAR

            fbTimerData();

(* Re-arm the zone retry while the answer is still outstanding. Doing it here
   rather than only on a result is the whole point: a request that was built and
   never answered would otherwise never be made again. *)
IF NOT bLocationKnown THEN
	fbLocationRetry.IN := TRUE;
END_IF
fbLocationRetry();

(* Every five minutes, publish everything again whether it moved or not, so a
   Home Assistant that reconnected still gets a value for a quiet sensor. *)
fbRepublish(IN := NOT fbRepublish.Q, PT := T#5M);
IF fbRepublish.Q THEN
	bRefreshDue := TRUE;

	(* Settings too. They are not retained either, and a setting changed from a
	   wall control rather than from Home Assistant would otherwise never be
	   noticed here. *)
	iSettingsCursor := 0;
	bSettingsDue := wSettingsMask <> 0;
END_IF

          

METHOD RequestBusTime : BOOL
                  IF NOT bNodeInitialized THEN	
	RequestBusTime := FALSE;
ELSIF fbTimerData.Q THEN
	RequestBusTime := TRUE;
ELSE
	RequestBusTime := FALSE;	
END_IF
                
END_METHOD

METHOD InitNode
  VAR_INPUT
    DeviceAddress : BYTE;
    NodeNumber : UINT;
    FriendlyName : STRING(GVL_MQTT.MQTT_SUFFIX_LEN);  (* Name of the room this component serves. Shown in Home Assistant; the topic keeps using the node number. *)
    DataPollingInterval : TIME;
  END_VAR
                  (* The measurements: read parameters 0..5, one frame. *)
THIS^.stStep.DeviceId		:= DeviceAddress;
THIS^.stStep.FunctionCode	:= 4;
THIS^.stStep.Address		:= (NodeNumber * 10) + 10;
THIS^.stStep.Quantity		:= 6;

(* The zone grouping: read parameter 9, on its own. Deliberately NOT folded into
   the step above by widening it to ten - 6, 7 and 8 are undefined on every
   component type and the box rejects a span that crosses them. *)
THIS^.stLocationStep.DeviceId		:= DeviceAddress;
THIS^.stLocationStep.FunctionCode	:= 4;
THIS^.stLocationStep.Address		:= (NodeNumber * 10) + 19;
THIS^.stLocationStep.Quantity		:= 1;

THIS^.FriendlyName := FriendlyName;
THIS^.fbTimerData.PT := DataPollingInterval;

(* The zone is asked for once and then left alone, so this only governs how
   long a lost answer goes unnoticed. Deliberately slow: it is a value that
   changes when somebody re-pairs the network and at no other time. *)
THIS^.fbLocationRetry.PT := T#30S;
THIS^.fbLocationRetry.IN := TRUE;
THIS^.NodeNumber := NodeNumber + 1;

THIS^.fbTimerData.IN := TRUE;

THIS^.bNodeInitialized := TRUE;

                
END_METHOD

METHOD InitMqtt
  VAR_INPUT
    MQTTPublishPrefix : POINTER TO STRING;
    MqttPublishTopicSuffix : STRING(255);
    pMqttPublishQueue : POINTER TO FB_MQTT_PUBLISH_QUEUE;
  END_VAR
                  THIS^.psMqttPublishTopicPrefix := MQTTPublishPrefix;
THIS^.MqttPublishTopicSuffix := MqttPublishTopicSuffix;
THIS^.pMqttPublishQueue := pMqttPublishQueue;

THIS^.bInitMqttDone := TRUE;
                
END_METHOD

METHOD PubMqttMessage
  VAR_INPUT
    Suffix : STRING(100);
    Data : STRING(100);
  END_VAR
                  IF bInitMqttDone THEN
		pMqttPublishQueue^.AddMessageOn(Lane := GVL_MQTT.MQTT_LANE_RS485,
			Payload := Data,
			Topic := CONCAT(CONCAT(CONCAT(CONCAT(psMqttPublishTopicPrefix^, MqttPublishTopicSuffix), '/'), UINT_TO_STRING(NodeNumber)), Suffix ),
			Qos := MQTT.QoS.ExactlyOnce,
			MqttRetain := FALSE
		);
END_IF
                
END_METHOD

METHOD OnStepResult
  VAR_INPUT
    Failed : BOOL;
    pData : POINTER TO A_RS485_READ_BUFFER;
    Count : INT;
  END_VAR
                  THIS^.fbTimerData.IN := TRUE;

IF Failed OR Count < 6 THEN
	RETURN;
END_IF

(* Read parameter 0 is the module type, and it decides what the other five mean.
   Resolving it here, once per read, is what stops the publisher guessing: on a
   window ventilator and an actuator board parameter 3 is the OUTDOOR temperature,
   and on an actuator board parameter 4 is a PWM duty cycle rather than CO2. *)
IF F_DUCO_NODE_TYPE(pData^[0]) <> THIS^.eType THEN
	THIS^.eType := F_DUCO_NODE_TYPE(pData^[0]);

	(* Duco assigns node numbers when components are paired, so a type that changes
	   under a node number is a real event and not a glitch: the zone has to be
	   asked for again, and Home Assistant has to be told what this node now is. *)
	(* Clearing this re-opens the question; the retry clock in the body does the
	   asking. RequestLocation ignores an Unknown type on its own. *)
	THIS^.bLocationKnown	:= FALSE;
	THIS^.uiLocationTries	:= 0;
	THIS^.bAnnounced		:= FALSE;
	(* What is writable depends on what the component is, so the settings sweep
	   is re-armed from scratch here as well. *)
	THIS^.wSettingsMask	:= THIS^.SettingsMaskFor(eT := THIS^.eType);
	THIS^.iSettingsCursor	:= 0;
	THIS^.bSettingsDue		:= THIS^.wSettingsMask <> 0;

	PubMqttMessage(Suffix := '/TYPE', Data := F_DUCO_TYPE_TEXT(THIS^.eType));
END_IF

(* Publish only what changed. Topics are not retained, so a value that never
   moves would never reach a reconnecting Home Assistant - hence the periodic
   refresh that forces a full publish regardless. *)
bChanged := NOT bPublishedOnce OR bRefreshDue;
FOR iChk := 0 TO 5 DO
	IF pData^[iChk] <> awLastRaw[iChk] THEN
		bChanged := TRUE;
	END_IF
	awLastRaw[iChk] := pData^[iChk];
END_FOR

IF bChanged THEN
	bPublishedOnce := TRUE;
	bRefreshDue := FALSE;
	THIS^.PublishDecoded(pData := pData, Count := Count);
END_IF

                
END_METHOD

METHOD GetStep : ST_RS485_STEP
                  (* Clearing the timer here rather than in RequestBusTime is what keeps that
   method a pure predicate - the parent, and through it the scheduler, may ask
   more than once per cycle. *)
IF fbTimerData.Q THEN
	THIS^.fbTimerData.IN := FALSE;
	GetStep := THIS^.stStep;
END_IF

                
END_METHOD

(* TRUE while this node still owes its zone number. See GetLocationStep. *)
METHOD RequestLocation : BOOL
                  (* Pure predicate, like RequestBusTime - the parent, and through it the
   scheduler, may ask more than once per cycle. Every side effect lives in
   GetLocationStep and in the body. *)
RequestLocation := bNodeInitialized
			AND NOT bLocationKnown
			AND (uiLocationTries < 3)
			AND (eType <> E_RS485_DUCO_NODE_TYPE.Unknown)
			AND fbLocationRetry.Q;

                
END_METHOD

(* The zone read, for the parent to put into a transaction it is building. *)
METHOD GetLocationStep : ST_RS485_STEP
                  (* Clearing the clock here rather than in RequestLocation is what keeps that
   method a pure predicate. Returns a zero-filled step if the clock has lapsed
   since the caller asked - the caller checks Quantity before using it. *)
IF fbLocationRetry.Q THEN
	THIS^.fbLocationRetry.IN := FALSE;
	THIS^.uiLocationTries := THIS^.uiLocationTries + 1;
	GetLocationStep := THIS^.stLocationStep;
END_IF

                
END_METHOD

(* Result of the zone read. Called by the parent, which owns the step map. *)
METHOD OnLocationResult
  VAR_INPUT
    Failed : BOOL;
    pData : POINTER TO A_RS485_READ_BUFFER;
    Count : INT;
  END_VAR
                  IF NOT Failed AND Count >= 1 THEN
	THIS^.bLocationKnown := TRUE;
	PubMqttMessage(Suffix := '/ZONE', Data := WORD_TO_STRING(pData^[0]));
END_IF

(* A failure needs no action: bLocationKnown stays FALSE, the body re-arms the
   clock, and the read comes round again. *)

                
END_METHOD

(* Publish read parameters 1..5 under the names this node's type gives them. *)
METHOD PublishDecoded
  VAR_INPUT
    pData : POINTER TO A_RS485_READ_BUFFER;
    Count : INT;
  END_VAR
                  (* One branch per component class, because the same register carries different
   quantities on different components. Anything not named here publishes nothing:
   an unrecognised component gets its raw registers below and no labels. *)
CASE eType OF

E_RS485_DUCO_NODE_TYPE.ValveSensorless,
E_RS485_DUCO_NODE_TYPE.ValveCO2,
E_RS485_DUCO_NODE_TYPE.ValveHumidity,
E_RS485_DUCO_NODE_TYPE.ValveHumidityCO2:
	PubMqttMessage(Suffix := '/STATUS', Data := F_DUCO_STATUS_TEXT(pData^[1]));
	PubMqttMessage(Suffix := '/POS', Data := WORD_TO_STRING(pData^[2]));
	PubMqttMessage(Suffix := '/TEMP', Data := F_DUCO_SCALED_TEXT(WORD_TO_INT(pData^[3]), 10));
	IF eType = E_RS485_DUCO_NODE_TYPE.ValveCO2 OR eType = E_RS485_DUCO_NODE_TYPE.ValveHumidityCO2 THEN
		PubMqttMessage(Suffix := '/CO2', Data := WORD_TO_STRING(pData^[4]));
	END_IF
	IF eType = E_RS485_DUCO_NODE_TYPE.ValveHumidity OR eType = E_RS485_DUCO_NODE_TYPE.ValveHumidityCO2 THEN
		PubMqttMessage(Suffix := '/RH', Data := F_DUCO_SCALED_TEXT(WORD_TO_INT(pData^[5]), 100));
	END_IF

E_RS485_DUCO_NODE_TYPE.UserControl:
	PubMqttMessage(Suffix := '/STATUS', Data := F_DUCO_STATUS_TEXT(pData^[1]));
	PubMqttMessage(Suffix := '/POS', Data := WORD_TO_STRING(pData^[2]));
	(* A battery unit has no temperature sensor and answers 0. Published anyway:
	   there is no flag distinguishing the two, so suppressing it would need a
	   guess about which kind of wall control this is. *)
	PubMqttMessage(Suffix := '/TEMP', Data := F_DUCO_SCALED_TEXT(WORD_TO_INT(pData^[3]), 10));

E_RS485_DUCO_NODE_TYPE.SensorCO2:
	PubMqttMessage(Suffix := '/STATUS', Data := F_DUCO_STATUS_TEXT(pData^[1]));
	PubMqttMessage(Suffix := '/TEMP', Data := F_DUCO_SCALED_TEXT(WORD_TO_INT(pData^[3]), 10));
	PubMqttMessage(Suffix := '/CO2', Data := WORD_TO_STRING(pData^[4]));

E_RS485_DUCO_NODE_TYPE.SensorHumidity:
	PubMqttMessage(Suffix := '/STATUS', Data := F_DUCO_STATUS_TEXT(pData^[1]));
	PubMqttMessage(Suffix := '/TEMP', Data := F_DUCO_SCALED_TEXT(WORD_TO_INT(pData^[3]), 10));
	PubMqttMessage(Suffix := '/RH', Data := F_DUCO_SCALED_TEXT(WORD_TO_INT(pData^[5]), 100));

E_RS485_DUCO_NODE_TYPE.WindowVentilator:
	PubMqttMessage(Suffix := '/STATUS', Data := F_DUCO_STATUS_TEXT(pData^[1]));
	(* 0 shut, 100 open - an opening, not an extraction level, which is why it is
	   not published as POS alongside the valves. *)
	PubMqttMessage(Suffix := '/OPEN', Data := WORD_TO_STRING(pData^[2]));
	PubMqttMessage(Suffix := '/TEMP_OUT', Data := F_DUCO_SCALED_TEXT(WORD_TO_INT(pData^[3]), 10));

E_RS485_DUCO_NODE_TYPE.SwitchSensor:
	PubMqttMessage(Suffix := '/STATUS', Data := F_DUCO_STATUS_TEXT(pData^[1]));
	PubMqttMessage(Suffix := '/POS', Data := WORD_TO_STRING(pData^[2]));

E_RS485_DUCO_NODE_TYPE.ActuatorBoard:
	PubMqttMessage(Suffix := '/STATUS', Data := F_DUCO_STATUS_TEXT(pData^[1]));
	PubMqttMessage(Suffix := '/POS', Data := WORD_TO_STRING(pData^[2]));
	PubMqttMessage(Suffix := '/TEMP_OUT', Data := F_DUCO_SCALED_TEXT(WORD_TO_INT(pData^[3]), 10));
	(* Parameter 4 is the PWM duty cycle on this component, and CO2 on nearly every
	   other one. Publishing it as CO2 is the mistake the type branch prevents. *)
	PubMqttMessage(Suffix := '/PWM', Data := WORD_TO_STRING(pData^[4]));

ELSE
	(* Unknown type: the registers, unlabelled. Enough to identify a new component
	   from the broker without pretending to know what its numbers mean. *)
	PubMqttMessage(Suffix := '/read/0', Data := WORD_TO_STRING(pData^[0]));
	PubMqttMessage(Suffix := '/read/1', Data := WORD_TO_STRING(pData^[1]));
	PubMqttMessage(Suffix := '/read/2', Data := WORD_TO_STRING(pData^[2]));
	PubMqttMessage(Suffix := '/read/3', Data := WORD_TO_STRING(pData^[3]));
	PubMqttMessage(Suffix := '/read/4', Data := WORD_TO_STRING(pData^[4]));
	PubMqttMessage(Suffix := '/read/5', Data := WORD_TO_STRING(pData^[5]));
END_CASE

                
END_METHOD

(* What this node is, as last read off the bus. Unknown before the first answer. *)
METHOD GetNodeType : E_RS485_DUCO_NODE_TYPE
                  GetNodeType := THIS^.eType;

                
END_METHOD

METHOD GetFriendlyName : STRING(GVL_MQTT.MQTT_SUFFIX_LEN)
                  GetFriendlyName := THIS^.FriendlyName;

                
END_METHOD

METHOD GetNodeNumber : UINT
                  GetNodeNumber := THIS^.NodeNumber;

                
END_METHOD

METHOD NeedsAnnounce : BOOL
                  (* Pure predicate. The parent sweeps every node with it each cycle. *)
NeedsAnnounce := bNodeInitialized
			AND NOT bAnnounced
			AND (eType <> E_RS485_DUCO_NODE_TYPE.Unknown);

                
END_METHOD

METHOD SetAnnounced
                  THIS^.bAnnounced := TRUE;

                
END_METHOD

(* Which registers of a component type hold a setting that is announced. One bit per register, bit n for register n. *)
METHOD SettingsMaskFor : WORD
  VAR_INPUT
    eT : E_RS485_DUCO_NODE_TYPE;
  END_VAR
                  (* Taken from what AnnounceNode actually announces, type by type: a register is
   in here exactly when some entity names it as a state topic. Register 9 is
   deliberately absent - it is the action, written by the buttons, and its
   result is reported under a different encoding in read parameter 1, so
   reading 9 back would say nothing an entity could use. *)
CASE eT OF
	(* The four valve types share an announce branch, so they share a mask. A
	   sensorless valve has no humidity or CO2 setpoint and will simply fail the
	   read for those registers, which publishes nothing - the same outcome as
	   before this existed. *)
	E_RS485_DUCO_NODE_TYPE.ValveSensorless,
	E_RS485_DUCO_NODE_TYPE.ValveCO2,
	E_RS485_DUCO_NODE_TYPE.ValveHumidity,
	E_RS485_DUCO_NODE_TYPE.ValveHumidityCO2:
		SettingsMaskFor := 16#007F;

	E_RS485_DUCO_NODE_TYPE.UserControl:
		SettingsMaskFor := 16#00F1;

	E_RS485_DUCO_NODE_TYPE.SensorCO2:
		SettingsMaskFor := 16#0003;

	E_RS485_DUCO_NODE_TYPE.SensorHumidity:
		SettingsMaskFor := 16#000D;

	E_RS485_DUCO_NODE_TYPE.WindowVentilator:
		SettingsMaskFor := 16#0071;

	E_RS485_DUCO_NODE_TYPE.SwitchSensor:
		SettingsMaskFor := 16#0007;

	E_RS485_DUCO_NODE_TYPE.ActuatorBoard:
		SettingsMaskFor := 16#0073;

ELSE
	(* Unknown, or a type nothing writable is announced for. *)
	SettingsMaskFor := 0;
END_CASE

                
END_METHOD

(* TRUE while a setting register still needs reading back. Pure predicate. *)
METHOD RequestSettings : BOOL
                  (* Pure, like RequestBusTime and RequestLocation: the parent may ask several
   times in one cycle, and the cursor is advanced by GetSettingsStep. *)
RequestSettings := FALSE;
IF NOT bSettingsDue OR wSettingsMask = 0 THEN
	RETURN;
END_IF

FOR iS := iSettingsCursor TO 9 DO
	IF (wSettingsMask AND SHL(WORD#1, INT_TO_BYTE(iS))) <> 0 THEN
		RequestSettings := TRUE;
		RETURN;
	END_IF
END_FOR

                
END_METHOD

(* The next setting register to read back. Zero-filled when none is due; the caller checks Quantity before using it. *)
METHOD GetSettingsStep : ST_RS485_STEP
                  (* Advancing the cursor here, not in RequestSettings, is what keeps that a pure
   predicate - the same split GetStep and GetLocationStep use.

   The cursor moves past this register whether or not the read succeeds. A
   failed one is simply not published and is picked up by the next refresh;
   retrying inside the sweep would let one dead register stall the rest. *)
iSettingsPending := -1;

FOR iS := iSettingsCursor TO 9 DO
	IF (wSettingsMask AND SHL(WORD#1, INT_TO_BYTE(iS))) <> 0 THEN
		iSettingsPending := iS;
		iSettingsCursor := iS + 1;
		EXIT;
	END_IF
END_FOR

IF iSettingsPending >= 0 THEN
	(* Function 3: these are holding registers, written with function 6 and read
	   back from the same address. That pairing is proven on hardware. *)
	THIS^.stSettingsStep.DeviceId		:= THIS^.stStep.DeviceId;
	THIS^.stSettingsStep.FunctionCode	:= 3;
	THIS^.stSettingsStep.Address		:= (NodeNumber * 10) + INT_TO_UINT(iSettingsPending);
	THIS^.stSettingsStep.Quantity		:= 1;
	GetSettingsStep := THIS^.stSettingsStep;
END_IF

                
END_METHOD

(* A setting register came back. Publishes it on the topic its entity reads. *)
METHOD OnSettingsResult
  VAR_INPUT
    Failed : BOOL;
    pData : POINTER TO A_RS485_READ_BUFFER;
    Count : INT;
  END_VAR
                  (* Signed, not raw: -1 is how a Ducobox reports 'not overriding', and the entity
   is announced with a minimum of -1 to match. WORD_TO_STRING would publish
   65535 there. Every other value in range is identical either way. *)
IF NOT Failed AND Count >= 1 AND iSettingsPending >= 0 THEN
	PubMqttMessage(
		Suffix := CONCAT('/write/', INT_TO_STRING(iSettingsPending)),
		Data := INT_TO_STRING(WORD_TO_INT(pData^[0])));
END_IF

iSettingsPending := -1;

(* Done once the cursor is past the last set bit. RequestSettings answers FALSE
   from then on, until a refresh re-arms it. *)
IF NOT THIS^.RequestSettings() THEN
	bSettingsDue := FALSE;
END_IF

                
END_METHOD
END_FUNCTION_BLOCK

{attribute 'reflection'}
FUNCTION_BLOCK FB_RS485_EASTRON_SDM_POWER_MQTT EXTENDS FB_MQTT_BASE IMPLEMENTS I_RS485_DEVICE
  VAR
    {attribute 'noinit'}
    {attribute 'instance-path'}
    sInstancePath : STRING(GVL_MQTT.MQTT_TOPIC_LEN);  (* object's full instance name *)
    bStartup : BOOL := TRUE;
    fbTimerData : TON;
    bIsDataUpdated : BOOL := FALSE;
    DeviceType : E_RS485_EASTRON_SDM_DEVICE;
    stStepSmallMeter : ST_RS485_STEP;  (* Active power sits at a different input register on the single-phase meters than on the SDM630, so the step to send depends on DeviceType. Both are filled by FB_init in code - a declaration initialiser here could not be revised by a script afterwards. *)
    stStepSDM630 : ST_RS485_STEP;
  END_VAR
  VAR_OUTPUT
    ACTIVEPOWER : REAL := 0;
    DataAvailable : BOOL := FALSE;
    Error : BOOL := FALSE;
  END_VAR
  VAR
    fbMqttDiscoveryDevice : FB_EASTRON_SDM_MQTT_DISCOVERY_DEVICE;  (* The meter as a Home Assistant device of its own. This block reads one value, so the device carries a single sensor entity - but it still wants to be a device rather than a loose entity on the PLC, because the model and the availability topic belong to the meter, not to the controller. *)
  END_VAR

            (* --- self-wiring prologue ----------------------------------------------------
   Makes the InitMqtt and InitMqttDiscovery calls optional. Set FriendlyName at
   the declaration site and this block wires itself from GVL_MQTT on its
   first cyclic call, then announces itself to Home Assistant.

   Deliberately in the body rather than in FB_init: it dereferences GVL members
   and reads the reflection instance path, and doing that during initialisation
   would rely on an ordering nothing enforces and the compiler cannot check.

   The model this meter announces itself as is derived from DeviceType, which
   FB_init settles before the first cycle - so unlike the earlier InitRS485
   arrangement there is nothing here to wait for.

   Dormant while FriendlyName is empty, so existing projects and existing call
   sites keep working untouched. A block wired this way MUST be called
   cyclically, and nothing warns if it is not. *)
IF FriendlyName <> '' THEN

	IF NOT bInitMqttDone THEN
		THIS^.InitMqtt(
			MQTTPublishPrefix := ADR(GVL_MQTT.MqttPubRS485Prefix),
			pMqttPublishQueue := ADR(GVL_MQTT.fbMqttPublishQueue));
	END_IF

	IF bInitMqttDone AND NOT bInitMqttDiscoveryDone THEN
		THIS^.InitMqttDiscovery(
			Device := ADR(THIS^.fbMqttDiscoveryDevice),
			DeviceName := FriendlyName);
	END_IF

END_IF

fbTimerData();

IF bIsDataUpdated THEN
	bIsDataUpdated := FALSE;

	PubMqttMessage(Suffix := '/ACTP', Data := REAL_TO_STRING(ACTIVEPOWER));
END_IF

          

METHOD FB_init : BOOL
  VAR_INPUT
    bInitRetains : BOOL;  (* TRUE: the retain variables are initialized (reset warm / reset cold) *)
    bInCopyCode : BOOL;  (* TRUE: the instance will be copied to the copy code afterward (online change) *)
    DeviceAddress : BYTE;
    DeviceType : E_RS485_EASTRON_SDM_DEVICE;
    DataPollingInterval : TIME;
  END_VAR
                  (* Modbus address, meter model and poll rate all describe the wiring rather than
   a mode, so they are fixed for the life of the instance and belong here rather
   than in a runtime setter. Note the consequence: changing any of them
   afterwards means editing the declaration in the IDE - CODESYS stores an
   instance's FB_init arguments beside the declaration text, where no script can
   reach them.

   DeviceType decides which register is read, and it is also the model this block
   announces itself to Home Assistant as. Setting it here means both are settled
   before the first cycle, so the discovery config cannot be published against a
   model that has not been chosen yet. *)
THIS^.stStepSmallMeter.DeviceId		:= DeviceAddress;
THIS^.stStepSmallMeter.FunctionCode	:= 4;
THIS^.stStepSmallMeter.Address		:= 12;	(* SDM120 / SDM220 active power *)
THIS^.stStepSmallMeter.Quantity		:= 2;

THIS^.stStepSDM630.DeviceId		:= DeviceAddress;
THIS^.stStepSDM630.FunctionCode	:= 4;
THIS^.stStepSDM630.Address		:= 52;	(* SDM630 total active power *)
THIS^.stStepSDM630.Quantity		:= 2;

THIS^.DeviceType := DeviceType;

THIS^.fbTimerData.PT := DataPollingInterval;
THIS^.fbTimerData.IN := TRUE;

FB_init := TRUE;

                
END_METHOD

METHOD InitMqtt
  VAR_INPUT
    MQTTPublishPrefix : POINTER TO STRING;
    pMqttPublishQueue : POINTER TO FB_MQTT_PUBLISH_QUEUE;
  END_VAR
                  SUPER^._sInstancePath := THIS^.sInstancePath; // Due to reflection its location is important

(*pass trough*)
THIS^.pMqttPublishQueue := pMqttPublishQueue;
THIS^.psMqttPublishTopicPrefix := MQTTPublishPrefix;
SUPER^.InitBaseMqtt();
                
END_METHOD

METHOD PubMqttMessage
  VAR_INPUT
    Suffix : STRING(100);
    Data : STRING(100);
  END_VAR
                  IF bInitMqttDone THEN
		pMqttPublishQueue^.AddMessageOn(Lane := GVL_MQTT.MQTT_LANE_RS485,
			Payload := Data,
			Topic := CONCAT(THIS^.sMQTTPublishTopic, Suffix),
			Qos := MQTT.QoS.ExactlyOnce,
			MqttRetain := FALSE
		);
END_IF
                
END_METHOD

METHOD HasWork : E_RS485_WORK_LEVEL
                  (* Predicate only - the scheduler calls this on every device every cycle, and
   twice when it is looking for commands first. Nothing here may change state. *)
IF fbTimerData.Q THEN
	HasWork := E_RS485_WORK_LEVEL.POLL;
ELSE
	HasWork := E_RS485_WORK_LEVEL.NONE;
END_IF

                
END_METHOD

METHOD BuildTransaction : INT
  VAR_INPUT
    pSteps : POINTER TO A_RS485_STEP_LIST;
  END_VAR
  VAR
    iN : INT;
  END_VAR
                  BuildTransaction := 0;

IF fbTimerData.Q THEN
	fbTimerData.IN := FALSE;

	IF DeviceType = E_RS485_EASTRON_SDM_DEVICE.SDM630 THEN
		pSteps^[0]			:= stStepSDM630;
		BuildTransaction	:= 1;
	ELSIF DeviceType = E_RS485_EASTRON_SDM_DEVICE.SDM120
	   OR DeviceType = E_RS485_EASTRON_SDM_DEVICE.SDM220 THEN
		pSteps^[0]			:= stStepSmallMeter;
		BuildTransaction	:= 1;
	END_IF
	(* An unset DeviceType returns 0: the scheduler releases the bus and moves
	   on rather than sending a frame nobody asked for. *)
END_IF

                
END_METHOD

METHOD OnStepResult
  VAR_INPUT
    StepIndex : INT;
    Failed : BOOL;
    pData : POINTER TO A_RS485_READ_BUFFER;
    Count : INT;
  END_VAR
                  THIS^.Error := Failed;
THIS^.fbTimerData.IN := TRUE;

IF NOT Failed AND Count >= 2 THEN
	THIS^.ACTIVEPOWER := F_SWAP_WORDS_TO_REAL(pData^[0], pData^[1]);
	THIS^.DataAvailable := TRUE;
	THIS^.bIsDataUpdated := TRUE;
END_IF

                
END_METHOD

METHOD OnTransactionDone
  VAR_INPUT
    StepsRun : INT;
    Failures : INT;
  END_VAR
                  (* One announcement per transaction, at the point the bus is released. *)
IF StepsRun > 0 AND Failures >= StepsRun THEN
	PubMqttMessage(Suffix := '/availability', Data := 'offline');
ELSIF StepsRun > 0 THEN
	PubMqttMessage(Suffix := '/availability', Data := 'online');
END_IF

                
END_METHOD

METHOD InitMqttDiscovery
  VAR_INPUT
    Device : POINTER TO FB_EASTRON_SDM_MQTT_DISCOVERY_DEVICE;
    DeviceName : STRING(50);
    Model : STRING(20) := '';
    overruleId : STRING(255) := '';
  END_VAR
  VAR
    id : STRING(255);
    sResolvedModel : STRING(20);
  END_VAR
                  (* Announces the meter as a device carrying one sensor: active power. Unlike the
   SDM220 and SDM630 blocks this one serves three meter models, so the model
   string is derived from DeviceType rather than fixed - InitRS485 must therefore
   have run before this does, which is what the self-wiring prologue waits for.
   Pass Model explicitly to overrule the derivation. *)
IF bInitMqttDone AND NOT bInitMqttDiscoveryDone THEN

	IF Model <> '' THEN
		sResolvedModel := Model;
	ELSE
		CASE DeviceType OF
			E_RS485_EASTRON_SDM_DEVICE.SDM120:	sResolvedModel := 'SDM120';
			E_RS485_EASTRON_SDM_DEVICE.SDM220:	sResolvedModel := 'SDM220';
			E_RS485_EASTRON_SDM_DEVICE.SDM630:	sResolvedModel := 'SDM630';
		ELSE
			sResolvedModel := 'unknown';
		END_CASE
	END_IF

	id := SUPER^.ResolveEntityId(overruleId := overruleId);

	Device^.initEastronDevice(
		name := DeviceName,
		id := id,
		Model := sResolvedModel,
		availabilityTopic1 := GVL_MQTT.MqttAvailabilityTopic,
		availabilityTopic2 := CONCAT(THIS^.sMQTTPublishTopic, '/availability'),
		availabilityOnline := GVL_MQTT.MqttAvailabilityOnlinePayload,
		availabilityOffline := GVL_MQTT.MqttAvailabilityOfflinePayload,
		MqttDiscoveryPrefix := GVL_MQTT.MqttHADiscoveryPrefix,
		MqttDiagnosticTopic := CONCAT(THIS^.sMQTTPublishTopic, '/diagnostic'),
		pMqttPublishQueue := ADR(GVL_MQTT.fbMqttPublishQueue));

(* This device publishes from the RS485 task, so its messages take that
   task's queue lane. A lane may only ever have one producing task. *)
Device^.SetLane(Lane := GVL_MQTT.MQTT_LANE_RS485);

	Device^.CreateSensorEntity(
		Name := 'Active Power',
		Id := CONCAT(id, '_ACTP'),
		StateTopic := CONCAT(THIS^.sMQTTPublishTopic, '/ACTP'),
		DeviceClass := 'power',
		StateClass := 'measurement',
		UnitOfMeasurement := 'W');

	bInitMqttDiscoveryDone := TRUE;
END_IF

                
END_METHOD

(* Nothing to commission on this device. See I_RS485_DEVICE.GetCommissioning. *)
METHOD GetCommissioning : BOOL
  VAR_INPUT
    BusBaudrate : UDINT;
    pRequest : POINTER TO ST_RS485_COMMISSION_REQUEST;
  END_VAR
                  (* Nothing to commission. This device is configured on the device itself - switches,
   a display, or a factory setting that already matches this bus - so it answers at
   whatever the bus runs at and there is nothing for the commissioner to write.

   Which is the ordinary case: the cost of the whole mechanism, for a device like
   this one, is this method call once at bStartup. *)
GetCommissioning := FALSE;

                
END_METHOD
END_FUNCTION_BLOCK

{attribute 'reflection'}
FUNCTION_BLOCK FB_RS485_EASTRON_SDM220_MQTT EXTENDS FB_MQTT_BASE IMPLEMENTS I_RS485_DEVICE
  VAR
    {attribute 'noinit'}
    {attribute 'instance-path'}
    sInstancePath : STRING(GVL_MQTT.MQTT_TOPIC_LEN);  (* object's full instance name *)
    bStartup : BOOL := TRUE;
    astSteps : ARRAY[0..2] OF ST_RS485_STEP;  (* The three register blocks this meter is read in. Filled by FB_init in code rather than by a declaration initialiser: a value inside an existing structured initialiser cannot be changed from a script afterwards - the compiler goes on reading the stored structValue - and a register map is exactly the sort of thing somebody will want to change. *)
    aiStepMap : ARRAY[0..2] OF INT;  (* Which block each step of the current transaction was built from. The scheduler hands StepIndex back and nothing else, so this is what tells OnStepResult that step 1 is the frequency block and not the voltage block. It replaces the old ActiveRtuQuery tag, which had to be set in GetRtuQuery and cleared in ProcessDataArray to mean anything. *)
    fbTimerData : TON;  (* One timer for the whole meter. There used to be three, one per register block, which put a technicality of the SDM220's 40-register reply limit into the caller's hands: three intervals to choose, for one meter that is read all at once. *)
    bUpdate1 : BOOL := FALSE;
    bUpdate2 : BOOL := FALSE;
    bUpdate3 : BOOL := FALSE;
  END_VAR
  VAR_OUTPUT
    VOLTAGE : REAL := 0;
    CURRENT : REAL := 0;
    ACTIVEPOWER : REAL := 0;
    APPARENT_POWER : REAL := 0;
    REACTIVE_POWER : REAL := 0;
    POWER_FACTOR : REAL := 0;
    PHASE_ANGLE : REAL := 0;
    DataAvailable1 : BOOL := FALSE;
    Error1 : BOOL := FALSE;
    FREQUENCY : REAL := 0;
    IMPORT_ACTIVE_ENERGY : REAL := 0;
    EXPORT_ACTIVE_ENERGY : REAL := 0;
    IMPORT_REACTIVE_ENERGY : REAL := 0;
    EXPORT_REACTIVE_ENERGY : REAL := 0;
    DataAvailable2 : BOOL := FALSE;
    Error2 : BOOL := FALSE;
    TOTAL_ACTIVE_ENERGY : REAL := 0;
    TOTAL_REACTIVE_ENERGY : REAL := 0;
    DataAvailable3 : BOOL := FALSE;
    Error3 : BOOL := FALSE;
  END_VAR
  VAR
    fbMqttDiscoveryDevice : FB_EASTRON_SDM_MQTT_DISCOVERY_DEVICE;  (* The meter announced to Home Assistant as a device of its own, so its fourteen measurements group under one card instead of scattering across the PLC device. One per meter and its lifetime is the meter's, so it lives here rather than in a GVL - the SDM630 does the same. *)
  END_VAR

            (* --- self-wiring prologue ----------------------------------------------------
   Makes the InitMqtt and InitMqttDiscovery calls optional. Set FriendlyName at
   the declaration site and this block wires itself from GVL_MQTT on its
   first cyclic call, then announces itself to Home Assistant.

   Deliberately in the body rather than in FB_init: it dereferences GVL members
   and reads the reflection instance path, and doing that during initialisation
   would rely on an ordering nothing enforces and the compiler cannot check.

   Dormant while FriendlyName is empty, so existing projects and existing call
   sites keep working untouched.

   A block wired this way MUST be called cyclically. An instance whose body never
   runs is unwired and absent from Home Assistant, and nothing warns about that. *)
IF FriendlyName <> '' THEN

	IF NOT bInitMqttDone THEN
		THIS^.InitMqtt(
			MQTTPublishPrefix := ADR(GVL_MQTT.MqttPubRS485Prefix),
			pMqttPublishQueue := ADR(GVL_MQTT.fbMqttPublishQueue));
	END_IF

	IF bInitMqttDone AND NOT bInitMqttDiscoveryDone THEN
		THIS^.InitMqttDiscovery(
			Device := ADR(THIS^.fbMqttDiscoveryDevice),
			DeviceName := FriendlyName);
	END_IF

END_IF

fbTimerData();

(* Published through PubMqttMessage rather than by building each topic inline.
   The inline form concatenated the prefix and suffix at every one of these
   fourteen call sites, which is the same string sMQTTPublishTopic already holds -
   and the discovery configs advertise sMQTTPublishTopic. Two ways of spelling one
   topic is how a state topic and its discovery config drift apart. *)
IF bUpdate1 THEN
	bUpdate1 := FALSE;
	DataAvailable1 := TRUE;

	PubMqttMessage(Suffix := '/VOLT', Data := REAL_TO_STRING(VOLTAGE));
	PubMqttMessage(Suffix := '/CURR', Data := REAL_TO_STRING(CURRENT));
	PubMqttMessage(Suffix := '/ACTP', Data := REAL_TO_STRING(ACTIVEPOWER));
	PubMqttMessage(Suffix := '/APPP', Data := REAL_TO_STRING(APPARENT_POWER));
	PubMqttMessage(Suffix := '/REAP', Data := REAL_TO_STRING(REACTIVE_POWER));
	PubMqttMessage(Suffix := '/POWF', Data := REAL_TO_STRING(POWER_FACTOR));
	PubMqttMessage(Suffix := '/PHAA', Data := REAL_TO_STRING(PHASE_ANGLE));
END_IF

IF bUpdate2 THEN
	bUpdate2 := FALSE;
	DataAvailable2 := TRUE;

	PubMqttMessage(Suffix := '/FREQ', Data := REAL_TO_STRING(FREQUENCY));
	PubMqttMessage(Suffix := '/IMAE', Data := REAL_TO_STRING(IMPORT_ACTIVE_ENERGY));
	PubMqttMessage(Suffix := '/EXAE', Data := REAL_TO_STRING(EXPORT_ACTIVE_ENERGY));
	PubMqttMessage(Suffix := '/IMRE', Data := REAL_TO_STRING(IMPORT_REACTIVE_ENERGY));
	PubMqttMessage(Suffix := '/EXRE', Data := REAL_TO_STRING(EXPORT_REACTIVE_ENERGY));
END_IF

IF bUpdate3 THEN
	bUpdate3 := FALSE;
	DataAvailable3 := TRUE;

	PubMqttMessage(Suffix := '/TOTAE', Data := REAL_TO_STRING(TOTAL_ACTIVE_ENERGY));
	PubMqttMessage(Suffix := '/TOTRE', Data := REAL_TO_STRING(TOTAL_REACTIVE_ENERGY));
END_IF

          

METHOD InitMqtt
  VAR_INPUT
    MQTTPublishPrefix : POINTER TO STRING;
    pMqttPublishQueue : POINTER TO FB_MQTT_PUBLISH_QUEUE;
  END_VAR
                  SUPER^._sInstancePath := THIS^.sInstancePath; // Due to reflection its location is important

(*pass trough*)
THIS^.pMqttPublishQueue := pMqttPublishQueue;
THIS^.psMqttPublishTopicPrefix := MQTTPublishPrefix;
SUPER^.InitBaseMqtt();
                
END_METHOD

METHOD PubMqttMessage
  VAR_INPUT
    Suffix : STRING(100);
    Data : STRING(100);
  END_VAR
                  IF bInitMqttDone THEN
		pMqttPublishQueue^.AddMessageOn(Lane := GVL_MQTT.MQTT_LANE_RS485,
			Payload := Data,
			Topic := CONCAT(THIS^.sMQTTPublishTopic, Suffix),
			Qos := MQTT.QoS.ExactlyOnce,
			MqttRetain := FALSE
		);
END_IF
                
END_METHOD

METHOD HasWork : E_RS485_WORK_LEVEL
                  (* Predicate only - the scheduler calls this on every device every cycle, and
   twice when it is looking for commands first. Nothing here may change state. *)
IF fbTimerData.Q THEN
	HasWork := E_RS485_WORK_LEVEL.POLL;
ELSE
	HasWork := E_RS485_WORK_LEVEL.NONE;
END_IF

                
END_METHOD

METHOD BuildTransaction : INT
  VAR_INPUT
    pSteps : POINTER TO A_RS485_STEP_LIST;
  END_VAR
                  (* The whole meter in one grant of the bus. Three register blocks used to mean
   winning the bus three separate times, with every other device's traffic in
   between; and while they were separately timed, which of the three were due
   varied from round to round. They now always go together.

   aiStepMap records which block each step came from, because OnStepResult is told
   the step index and nothing else. *)
IF fbTimerData.Q THEN
	fbTimerData.IN := FALSE;

	pSteps^[0] := astSteps[0];		aiStepMap[0] := 1;
	pSteps^[1] := astSteps[1];		aiStepMap[1] := 2;
	pSteps^[2] := astSteps[2];		aiStepMap[2] := 3;

	BuildTransaction := 3;
ELSE
	BuildTransaction := 0;
END_IF

                
END_METHOD

METHOD OnStepResult
  VAR_INPUT
    StepIndex : INT;
    Failed : BOOL;
    pData : POINTER TO A_RS485_READ_BUFFER;
    Count : INT;
  END_VAR
                  IF StepIndex < 0 OR StepIndex > DINT_TO_INT(UPPER_BOUND(aiStepMap, 1)) THEN
	RETURN;
END_IF

(* Count is what actually came back, not what was asked for, so a short reply
   cannot be read past the end of. The timer is not re-armed here - see
   OnTransactionDone. *)
CASE aiStepMap[StepIndex] OF

1:	THIS^.Error1 := Failed;
	IF NOT Failed AND Count >= 38 THEN
		THIS^.VOLTAGE			:= F_SWAP_WORDS_TO_REAL(pData^[0], pData^[1]);
		THIS^.CURRENT			:= F_SWAP_WORDS_TO_REAL(pData^[6], pData^[7]);
		THIS^.ACTIVEPOWER		:= F_SWAP_WORDS_TO_REAL(pData^[12], pData^[13]);
		THIS^.APPARENT_POWER	:= F_SWAP_WORDS_TO_REAL(pData^[18], pData^[19]);
		THIS^.REACTIVE_POWER	:= F_SWAP_WORDS_TO_REAL(pData^[24], pData^[25]);
		THIS^.POWER_FACTOR		:= F_SWAP_WORDS_TO_REAL(pData^[30], pData^[31]);
		THIS^.PHASE_ANGLE		:= F_SWAP_WORDS_TO_REAL(pData^[36], pData^[37]);
		THIS^.bUpdate1 := TRUE;
	END_IF

2:	THIS^.Error2 := Failed;
	IF NOT Failed AND Count >= 10 THEN
		THIS^.FREQUENCY					:= F_SWAP_WORDS_TO_REAL(pData^[0], pData^[1]);
		THIS^.IMPORT_ACTIVE_ENERGY		:= F_SWAP_WORDS_TO_REAL(pData^[2], pData^[3]);
		THIS^.EXPORT_ACTIVE_ENERGY		:= F_SWAP_WORDS_TO_REAL(pData^[4], pData^[5]);
		THIS^.IMPORT_REACTIVE_ENERGY	:= F_SWAP_WORDS_TO_REAL(pData^[6], pData^[7]);
		THIS^.EXPORT_REACTIVE_ENERGY	:= F_SWAP_WORDS_TO_REAL(pData^[8], pData^[9]);
		THIS^.bUpdate2 := TRUE;
	END_IF

3:	THIS^.Error3 := Failed;
	IF NOT Failed AND Count >= 4 THEN
		THIS^.TOTAL_ACTIVE_ENERGY	:= F_SWAP_WORDS_TO_REAL(pData^[0], pData^[1]);
		THIS^.TOTAL_REACTIVE_ENERGY	:= F_SWAP_WORDS_TO_REAL(pData^[2], pData^[3]);
		THIS^.bUpdate3 := TRUE;
	END_IF

END_CASE

                
END_METHOD

METHOD OnTransactionDone
  VAR_INPUT
    StepsRun : INT;
    Failures : INT;
  END_VAR
                  (* One announcement per transaction, and one re-arm of the timer.

   The re-arm belongs here rather than in OnStepResult because a step skipped by
   an AbortOnError predecessor is never reported, and a meter that has stopped
   answering must still be retried. OnTransactionDone always runs. *)
fbTimerData.IN := TRUE;

IF StepsRun > 0 AND Failures >= StepsRun THEN
	PubMqttMessage(Suffix := '/availability', Data := 'offline');
ELSIF StepsRun > 0 THEN
	PubMqttMessage(Suffix := '/availability', Data := 'online');
END_IF

                
END_METHOD

METHOD InitMqttDiscovery
  VAR_INPUT
    Device : POINTER TO FB_EASTRON_SDM_MQTT_DISCOVERY_DEVICE;
    DeviceName : STRING(50);
    Model : STRING(20) := 'SDM220';
    overruleId : STRING(255) := '';
  END_VAR
  VAR
    id : STRING(255);
  END_VAR
                  (* Announces the meter as a device of its own, then one sensor entity per
   measurement. StateClass is what puts the energy totals into the Home
   Assistant energy dashboard; the instantaneous values are 'measurement', and
   power factor and phase angle carry none because neither is meaningful to
   sum or average over time.

   The three kvarh counters use DeviceClass 'reactive_energy', which Home
   Assistant gained in 2025.9. On an older Home Assistant an unrecognised device
   class makes it reject the whole discovery config, so those three entities
   would not appear at all - the symptom is a missing entity, not a wrong one. *)
IF bInitMqttDone AND NOT bInitMqttDiscoveryDone THEN

	id := SUPER^.ResolveEntityId(overruleId := overruleId);

	Device^.initEastronDevice(
		name := DeviceName,
		id := id,
		Model := Model,
		availabilityTopic1 := GVL_MQTT.MqttAvailabilityTopic,
		availabilityTopic2 := CONCAT(THIS^.sMQTTPublishTopic, '/availability'),
		availabilityOnline := GVL_MQTT.MqttAvailabilityOnlinePayload,
		availabilityOffline := GVL_MQTT.MqttAvailabilityOfflinePayload,
		MqttDiscoveryPrefix := GVL_MQTT.MqttHADiscoveryPrefix,
		MqttDiagnosticTopic := CONCAT(THIS^.sMQTTPublishTopic, '/diagnostic'),
		pMqttPublishQueue := ADR(GVL_MQTT.fbMqttPublishQueue));

(* This device publishes from the RS485 task, so its messages take that
   task's queue lane. A lane may only ever have one producing task. *)
Device^.SetLane(Lane := GVL_MQTT.MQTT_LANE_RS485);

	(* --- register block 1: the instantaneous electrical values ------------- *)

	Device^.CreateSensorEntity(
		Name := 'Voltage',
		Id := CONCAT(id, '_VOLT'),
		StateTopic := CONCAT(THIS^.sMQTTPublishTopic, '/VOLT'),
		DeviceClass := 'voltage',
		StateClass := 'measurement',
		UnitOfMeasurement := 'V');

	Device^.CreateSensorEntity(
		Name := 'Current',
		Id := CONCAT(id, '_CURR'),
		StateTopic := CONCAT(THIS^.sMQTTPublishTopic, '/CURR'),
		DeviceClass := 'current',
		StateClass := 'measurement',
		UnitOfMeasurement := 'A');

	Device^.CreateSensorEntity(
		Name := 'Active Power',
		Id := CONCAT(id, '_ACTP'),
		StateTopic := CONCAT(THIS^.sMQTTPublishTopic, '/ACTP'),
		DeviceClass := 'power',
		StateClass := 'measurement',
		UnitOfMeasurement := 'W');

	Device^.CreateSensorEntity(
		Name := 'Apparent Power',
		Id := CONCAT(id, '_APPP'),
		StateTopic := CONCAT(THIS^.sMQTTPublishTopic, '/APPP'),
		DeviceClass := 'apparent_power',
		StateClass := 'measurement',
		UnitOfMeasurement := 'VA');

	Device^.CreateSensorEntity(
		Name := 'Reactive Power',
		Id := CONCAT(id, '_REAP'),
		StateTopic := CONCAT(THIS^.sMQTTPublishTopic, '/REAP'),
		DeviceClass := 'reactive_power',
		StateClass := 'measurement',
		UnitOfMeasurement := 'var');

	Device^.CreateSensorEntity(
		Name := 'Power Factor',
		Id := CONCAT(id, '_POWF'),
		StateTopic := CONCAT(THIS^.sMQTTPublishTopic, '/POWF'),
		DeviceClass := 'power_factor',
		UnitOfMeasurement := '');

	Device^.CreateSensorEntity(
		Name := 'Phase Angle',
		Id := CONCAT(id, '_PHAA'),
		StateTopic := CONCAT(THIS^.sMQTTPublishTopic, '/PHAA'),
		DeviceClass := '',
		UnitOfMeasurement := '°');

	(* --- register block 2: frequency and the four energy counters ---------- *)

	Device^.CreateSensorEntity(
		Name := 'Frequency',
		Id := CONCAT(id, '_FREQ'),
		StateTopic := CONCAT(THIS^.sMQTTPublishTopic, '/FREQ'),
		DeviceClass := 'frequency',
		StateClass := 'measurement',
		UnitOfMeasurement := 'Hz');

	Device^.CreateSensorEntity(
		Name := 'Import Active Energy',
		Id := CONCAT(id, '_IMAE'),
		StateTopic := CONCAT(THIS^.sMQTTPublishTopic, '/IMAE'),
		DeviceClass := 'energy',
		StateClass := 'total_increasing',
		UnitOfMeasurement := 'kWh');

	Device^.CreateSensorEntity(
		Name := 'Export Active Energy',
		Id := CONCAT(id, '_EXAE'),
		StateTopic := CONCAT(THIS^.sMQTTPublishTopic, '/EXAE'),
		DeviceClass := 'energy',
		StateClass := 'total_increasing',
		UnitOfMeasurement := 'kWh');

	Device^.CreateSensorEntity(
		Name := 'Import Reactive Energy',
		Id := CONCAT(id, '_IMRE'),
		StateTopic := CONCAT(THIS^.sMQTTPublishTopic, '/IMRE'),
		DeviceClass := 'reactive_energy',
		StateClass := 'total_increasing',
		UnitOfMeasurement := 'kvarh');

	Device^.CreateSensorEntity(
		Name := 'Export Reactive Energy',
		Id := CONCAT(id, '_EXRE'),
		StateTopic := CONCAT(THIS^.sMQTTPublishTopic, '/EXRE'),
		DeviceClass := 'reactive_energy',
		StateClass := 'total_increasing',
		UnitOfMeasurement := 'kvarh');

	(* --- register block 3: the totals -------------------------------------- *)

	Device^.CreateSensorEntity(
		Name := 'Total Active Energy',
		Id := CONCAT(id, '_TOTAE'),
		StateTopic := CONCAT(THIS^.sMQTTPublishTopic, '/TOTAE'),
		DeviceClass := 'energy',
		StateClass := 'total_increasing',
		UnitOfMeasurement := 'kWh');

	Device^.CreateSensorEntity(
		Name := 'Total Reactive Energy',
		Id := CONCAT(id, '_TOTRE'),
		StateTopic := CONCAT(THIS^.sMQTTPublishTopic, '/TOTRE'),
		DeviceClass := 'reactive_energy',
		StateClass := 'total_increasing',
		UnitOfMeasurement := 'kvarh');

	bInitMqttDiscoveryDone := TRUE;
END_IF

                
END_METHOD

METHOD FB_init : BOOL
  VAR_INPUT
    bInitRetains : BOOL;  (* TRUE: the retain variables are initialized (reset warm / reset cold) *)
    bInCopyCode : BOOL;  (* TRUE: the instance will be copied to the copy code afterward (online change) *)
    DeviceAddress : BYTE;
    DataPollingInterval : TIME;
  END_VAR
                  (* Modbus address and poll rate describe the wiring, not a mode, so they are
   fixed for the life of the instance and belong here rather than in a runtime
   setter. Note the consequence: changing either afterwards means editing the
   declaration in the IDE - CODESYS stores an instance's FB_init arguments beside
   the declaration text, where no script can reach them.

   ONE interval covers the whole meter. The SDM220 will not return more than 40
   registers in a reply and its measurements are not in one contiguous run, so
   reading it takes three requests - but that is a property of the meter, not a
   decision a caller should be asked to make. All three go out together as a
   single transaction, so they cost one turn of the bus rather than three. *)
THIS^.astSteps[0].DeviceId		:= DeviceAddress;
THIS^.astSteps[0].FunctionCode	:= 4;
THIS^.astSteps[0].Address		:= 0;	(* voltage through phase angle *)
THIS^.astSteps[0].Quantity		:= 40;

THIS^.astSteps[1].DeviceId		:= DeviceAddress;
THIS^.astSteps[1].FunctionCode	:= 4;
THIS^.astSteps[1].Address		:= 70;	(* frequency, import and export energy *)
THIS^.astSteps[1].Quantity		:= 10;

THIS^.astSteps[2].DeviceId		:= DeviceAddress;
THIS^.astSteps[2].FunctionCode	:= 4;
THIS^.astSteps[2].Address		:= 342;	(* totals *)
THIS^.astSteps[2].Quantity		:= 4;

THIS^.fbTimerData.PT := DataPollingInterval;
THIS^.fbTimerData.IN := TRUE;

FB_init := TRUE;

                
END_METHOD

(* Nothing to commission on this device. See I_RS485_DEVICE.GetCommissioning. *)
METHOD GetCommissioning : BOOL
  VAR_INPUT
    BusBaudrate : UDINT;
    pRequest : POINTER TO ST_RS485_COMMISSION_REQUEST;
  END_VAR
                  (* Nothing to commission. This device is configured on the device itself - switches,
   a display, or a factory setting that already matches this bus - so it answers at
   whatever the bus runs at and there is nothing for the commissioner to write.

   Which is the ordinary case: the cost of the whole mechanism, for a device like
   this one, is this method call once at bStartup. *)
GetCommissioning := FALSE;

                
END_METHOD
END_FUNCTION_BLOCK

